// TwinCAT 3 PLC project RRP_Palletizer_Project
// ProgramVersion: 3.1.4023.0
// libraries:
//   Tc2_Standard, * (Beckhoff Automation GmbH)
//   Tc2_System, * (Beckhoff Automation GmbH)
//   Tc3_Module, * (Beckhoff Automation GmbH)
// project tree:
//   DUTs/ stMachineState.TcDUT, stMotor.TcDUT, stPneumatic1.TcDUT, stPneumatic2.TcDUT
//   GVLs/ Data_GVL.TcGVL, HMI_GVL.TcGVL, InputOutput_GVL.TcGVL
//   / BoxTask.TcTTO
//   POUs/S01_Box/ EM01_BoxShorting.TcPOU, UN01_StateMachineBox.TcPOU
//   POUs/S02_Pallet/ EM01_Dispenser.TcPOU, EM02_Shuttle.TcPOU, EM03_PalletOutfeed.TcPOU, UN01_StateMachinePallet.TcPOU
//   POUs/S03_Robot_1/ EM03_PlacingArea_2.TcPOU, EM04_PlacingArea_3.TcPOU, EM05_PlacingArea_4.TcPOU, EM01_BoxInfeed.TcPOU, EM02_PlacingArea_1.TcPOU, EM06_Robot.TcPOU, UN01_StateMachineRobot_1.TcPOU
//   POUs/Functions Blocks/ BLINK.TcPOU, FB_StateManager.TcPOU, MotorManagement.TcPOU, Pneumatic_1Coil_Management.TcPOU, Pneumatic_2Coil_Management.TcPOU
// real-time tasks:
//   TASK PlcTask: cycle T#10ms, priority 20, ADS port 350
//   TASK Box: cycle T#10ms, priority 21, ADS port 351

CONFIGURATION RRP_Palletizer_Project
    RESOURCE PLC ON TwinCAT3
        TASK BoxTask(INTERVAL := T#10ms, PRIORITY := 21);
        PROGRAM UN01_StateMachineBox WITH BoxTask : UN01_StateMachineBox;
        PROGRAM EM01_BoxShorting WITH BoxTask : EM01_BoxShorting;
    END_RESOURCE
END_CONFIGURATION

// ---- DUTs/stMachineState.TcDUT
TYPE stMachineState :
STRUCT
	Error 		: BOOL;
	CheckSafety	: BOOL;
	Aborted		: BOOL;
	Initialize	: BOOL;
	CheckToRun	: BOOL;
	Ready		: BOOL;
	Running		: BOOL;
	Stopped		: BOOL;
	ManualMode	: BOOL;
END_STRUCT
END_TYPE

// ---- DUTs/stMotor.TcDUT
TYPE stMotor :	
STRUCT
	Name				: STRING;
	TestModeActive		: BOOL;
	UseReverse			: BOOL;
	iTestForward		: BOOL;
	iTestReverse		: BOOL;
	oMoveForward		: BOOL;
	oMoveReverse		: BOOL;
	oResetError			: BOOL;
	Status_MotorRunning	: BOOL;
	Status_Error		: BOOL;
	ErrorID				: UINT;
END_STRUCT
END_TYPE

// ---- DUTs/stPneumatic1.TcDUT
TYPE stPneumatic1 : //v1.0
// UDT untuk merepresentasikan faceplate pneumatic valve 1 coil
//	Changelog:
	(* 
	v1.0 [27.12.2021] Start development UDT - Fabrilian Asali	*)	


STRUCT
	Name: STRING;
	
	TestModeActive: BOOL;
	iTest: BOOL;
	
	iSensorRetract: BOOL;
	iSensorAdvanced: BOOL;
	
	oPneumatic: BOOL;
	
	Trigger_Retract: BOOL;
	Trigger_Advanced: BOOL;
	FB_DoneRetract: BOOL;
	FB_DoneAdvanced: BOOL;
	
	Error_Retract: BOOL;
	Error_Advanced: BOOL;
END_STRUCT
END_TYPE

// ---- DUTs/stPneumatic2.TcDUT
TYPE stPneumatic2 :	//v1.0
// UDT untuk merepresentasikan faceplate pneumatic valve 1 coil
//	Changelog:
	(* 
	v1.0 [27.12.2021] Start development UDT - Fabrilian Asali	*)	

STRUCT
	Name: STRING;
	
	TestModeActive: BOOL;
	iTestRetract: BOOL;
	iTestAdvanced: BOOL;
	
	iSensorRetract: BOOL;
	iSensorAdvanced: BOOL;
	
	oPneumaticRetract: BOOL;
	oPneumaticAdvanced: BOOL;
	
	Trigger_Retract: BOOL;
	Trigger_Advanced: BOOL;
	FB_DoneRetract: BOOL;
	FB_DoneAdvanced: BOOL;
	
	Error_Retract: BOOL;
	Error_Advanced: BOOL;
END_STRUCT
END_TYPE

// ---- GVLs/Data_GVL.TcGVL
{attribute 'qualified_only'}
VAR_GLOBAL
	
//-----Box----	
	//Shorting
	StateMachineShorting			: stMachineState;
	StateMachineShorting_Error		: BOOL;
	StateMachineShorting_ErrorMsg	: STRING;
	StateMachineShorting_stsMachine	: STRING;
	bFL_StartShorting				: BOOL;
	bFL_StopShorting				: BOOL;
	bFL_ResetShorting				: BOOL;
	bFL_AckShorting					: BOOL;
	bFL_MachineErrorShorting		: BOOL;
	bFL_AutoManuaModeShorting		: BOOL;
	
//-----Pallet----		
	//Dispenser
	StateMachineDispenser			: stMachineState;
	StateMachineDispenser_Error		: BOOL;
	StateMachineDispenser_ErrorMsg	: STRING;
	StateMachineDispenser_stsMachine: STRING;
	bFL_StartDispenser				: BOOL;
	bFL_StopDispenser				: BOOL;
	bFL_ResetDispenser				: BOOL;
	bFL_AckDispenser				: BOOL;
	bFL_MachineErrorDispenser		: BOOL;
	bFL_AutoManuaModeDispenser		: BOOL;
	//Shuttle
	StateMachineShuttle				: stMachineState;
	StateMachineShuttle_Error		: BOOL;
	StateMachineShuttle_ErrorMsg	: STRING;
	StateMachineShuttle_stsMachine	: STRING;
	bFL_StartShuttle				: BOOL;
	bFL_StopShuttle					: BOOL;
	bFL_ResetShuttle				: BOOL;
	bFL_AckShuttle					: BOOL;
	bFL_MachineErrorShuttle			: BOOL;
	bFL_AutoManuaModeShuttle		: BOOL;
	//Outfeed
	StateMachineOutfeed				: stMachineState;
	StateMachineOutfeed_Error		: BOOL;
	StateMachineOutfeed_ErrorMsg	: STRING;
	StateMachineOutfeed_stsMachine	: STRING;
	bFL_StartOutfeed				: BOOL;
	bFL_StopOutfeed					: BOOL;
	bFL_ResetOutfeed				: BOOL;
	bFL_AckOutfeed					: BOOL;
	bFL_MachineErrorOutfeed			: BOOL;
	bFL_AutoManuaModeOutfeed		: BOOL;
	
//-----Robot----		
	//Infeed
	StateMachineInfeed				: stMachineState;
	StateMachineInfeed_Error		: BOOL;
	StateMachineInfeed_ErrorMsg		: STRING;
	StateMachineInfeed_stsMachine	: STRING;
	bFL_StartInfeed					: BOOL;
	bFL_StopInfeed					: BOOL;
	bFL_ResetInfeed					: BOOL;
	bFL_AckInfeed					: BOOL;
	bFL_MachineErrorInfeed			: BOOL;
	bFL_AutoManuaModeInfeed			: BOOL;	
	//Placing_1
	StateMachinePlacing_1			: stMachineState;
	StateMachinePlacing_1_Error		: BOOL;
	StateMachinePlacing_1_ErrorMsg	: STRING;
	StateMachinePlacing_1_stsMachine: STRING;
	bFL_StartPlacing_1				: BOOL;
	bFL_StopPlacing_1				: BOOL;
	bFL_ResetPlacing_1				: BOOL;
	bFL_AckPlacing_1				: BOOL;
	bFL_MachineErrorPlacing_1		: BOOL;
	bFL_AutoManuaModePlacing_1		: BOOL;
	//Placing_2
	StateMachinePlacing_2			: stMachineState;
	StateMachinePlacing_2_Error		: BOOL;
	StateMachinePlacing_2_ErrorMsg	: STRING;
	StateMachinePlacing_2_stsMachine: STRING;
	bFL_StartPlacing_2				: BOOL;
	bFL_StopPlacing_2				: BOOL;
	bFL_ResetPlacing_2				: BOOL;
	bFL_AckPlacing_2				: BOOL;
	bFL_MachineErrorPlacing_2		: BOOL;
	bFL_AutoManuaModePlacing_2		: BOOL;
	//Placing_3
	StateMachinePlacing_3			: stMachineState;
	StateMachinePlacing_3_Error		: BOOL;
	StateMachinePlacing_3_ErrorMsg	: STRING;
	StateMachinePlacing_3_stsMachine: STRING;
	bFL_StartPlacing_3				: BOOL;
	bFL_StopPlacing_3				: BOOL;
	bFL_ResetPlacing_3				: BOOL;
	bFL_AckPlacing_3				: BOOL;
	bFL_MachineErrorPlacing_3		: BOOL;
	bFL_AutoManuaModePlacing_3		: BOOL;
	//Placing_4
	StateMachinePlacing_4			: stMachineState;
	StateMachinePlacing_4_Error		: BOOL;
	StateMachinePlacing_4_ErrorMsg	: STRING;
	StateMachinePlacing_4_stsMachine: STRING;
	bFL_StartPlacing_4				: BOOL;
	bFL_StopPlacing_4				: BOOL;
	bFL_ResetPlacing_4				: BOOL;
	bFL_AckPlacing_4				: BOOL;
	bFL_MachineErrorPlacing_4		: BOOL;
	bFL_AutoManuaModePlacing_4		: BOOL;
	//Robot
	StateMachineRobot				: stMachineState;
	StateMachineRobot_Error			: BOOL;
	StateMachineRobot_ErrorMsg		: STRING;
	StateMachineRobot_stsMachine	: STRING;
	bFL_StartRobot		 			: BOOL;
	bFL_StopRobot					: BOOL;
	bFL_ResetRobot					: BOOL;
	bFL_AckRobot					: BOOL;
	bFL_MachineErrorRobot			: BOOL;
	bFL_AutoManuaModeRobot			: BOOL;
	
	bStartButton 					: BOOL;
	bStopButton 					: BOOL;
	bResetButton 					: BOOL;
	bAckButton 						: BOOL;
	bEmergencyStop 					: BOOL;
END_VAR

// ---- GVLs/HMI_GVL.TcGVL
{attribute 'qualified_only'}
VAR_GLOBAL
//-----Box----
	//Shorting
	bTestModeEnableShorting	: BOOL;
	bStartButtonShorting	: BOOL;
	bStopButtonShorting		: BOOL;
	bResetButtonShorting	: BOOL;

//-----Pallet----
	//Dispenser
	bTestModeEnableDispenser: BOOL;
	bStartButtonDispenser	: BOOL;
	bStopButtonDispenser	: BOOL;
	bResetButtonDispenser	: BOOL;
	//Outfeed
	bTestModeEnableOutfeed	: BOOL;
	bStartButtonOutfeed		: BOOL;
	bStopButtonOutfeed		: BOOL;
	bResetButtonOutfeed		: BOOL;
	//Shuttle
	bTestModeEnableShuttle	: BOOL;
	bStartButtonShuttle		: BOOL;
	bStopButtonShuttle		: BOOL;
	bResetButtonShuttle		: BOOL;

//-----Robot----
	//Infeed
	bTestModeEnableInfeed	: BOOL;
	bStartButtonInfeed		: BOOL;
	bStopButtonInfeed		: BOOL;
	bResetButtonInfeed		: BOOL;
	//Placing_1
	bTestModeEnablePlacing_1: BOOL;
	bStartButtonPlacing_1	: BOOL;
	bStopButtonPlacing_1	: BOOL;
	bResetButtonPlacing_1	: BOOL;
	//Placing_2
	bTestModeEnablePlacing_2: BOOL;
	bStartButtonPlacing_2	: BOOL;
	bStopButtonPlacing_2	: BOOL;
	bResetButtonPlacing_2	: BOOL;
	//Placing_3
	bTestModeEnablePlacing_3: BOOL;
	bStartButtonPlacing_3	: BOOL;
	bStopButtonPlacing_3	: BOOL;
	bResetButtonPlacing_3	: BOOL;
	//Placing_4
	bTestModeEnablePlacing_4: BOOL;
	bStartButtonPlacing_4	: BOOL;
	bStopButtonPlacing_4	: BOOL;
	bResetButtonPlacing_4	: BOOL;
	//Robot
	bTestModeEnableRobot	: BOOL;
	bStartButtonRobot		: BOOL;
	bStopButtonRobot		: BOOL;
	bResetButtonRobot		: BOOL;
END_VAR

// ---- GVLs/InputOutput_GVL.TcGVL
{attribute 'qualified_only'}
VAR_GLOBAL
	//Panel 1
	//Digital Input 16 Point EL1809
	xIn1000				AT 		%I*			: BOOL;		// Push Button Run at Main Panel
	xIn1001				AT 		%I*			: BOOL;		// Push Button Stop at Main Panel
	xIn1002				AT 		%I*			: BOOL;		// Push Button Alarm Reset at Main Panel
	xIn1003				AT 		%I*			: BOOL;		// Push Button Acknowledge at Main Panel
	xIn1004				AT 		%I*			: BOOL;		// Auto/Manual Mode at Main Panel
	xIn1005				AT 		%I*			: BOOL;		// Emergency Stop at Main Panel
	xIn1006				AT 		%I*			: BOOL;		//	
	xIn1007				AT 		%I*			: BOOL;		//
	xIn1008				AT 		%I*			: BOOL;		//
	xIn1009				AT 		%I*			: BOOL;		//
	xIn1010				AT 		%I*			: BOOL;		//
	xIn1011				AT 		%I*			: BOOL;		//
	xIn1012				AT 		%I*			: BOOL;		//
	xIn1013				AT 		%I*			: BOOL;		//
	xIn1014				AT 		%I*			: BOOL;		//
	xIn1015				AT 		%I*			: BOOL;		// Pressure Switch
	//Digital Input 16 Point EL1809
	xIn1100				AT 		%I*			: BOOL;		// Feedback Barcoder Reading Conveyor is Running
	xIn1101				AT 		%I*			: BOOL;		// Feedback Box Infeed Roller Conveyor 1 is Running
	xIn1102				AT 		%I*			: BOOL;		// Feedback Box Infeed Roller Conveyor 2 is Running 
	xIn1103				AT 		%I*			: BOOL;		// Feedback Box Infeed Roller Conveyor 3 is Running
	xIn1104				AT 		%I*			: BOOL;		// Feedback Box Buffer Roller Conveyor 1 is Running
	xIn1105				AT 		%I*			: BOOL;		// Feedback Box Buffer Roller Conveyor 2 is Running
	xIn1106				AT 		%I*			: BOOL;		// Feedback Box Stop & Go Belt Conveyor is Running
	xIn1107				AT 		%I*			: BOOL;		// Feedback Box Picking Roller Conveyor is Running
	xIn1108				AT 		%I*			: BOOL;		//
	xIn1109				AT 		%I*			: BOOL;		//
	xIn1110				AT 		%I*			: BOOL;		//
	xIn1111				AT 		%I*			: BOOL;		//
	xIn1112				AT 		%I*			: BOOL;		//
	xIn1113				AT 		%I*			: BOOL;		//
	xIn1114				AT 		%I*			: BOOL;		//
	xIn1115				AT 		%I*			: BOOL;		// 
	//Digital Input 16 Point EL1809
	xIn1200				AT 		%I*			: BOOL;		// RSW to Check Pneu Box Pusher for Reject Barcode when Rtc
	xIn1201				AT 		%I*			: BOOL;		// RSW to Check Pneu Box Pusher for Reject Barcode when Adv
	xIn1202				AT 		%I*			: BOOL;		// RSW to Check Pneu Box Pusher for Reject Weight when Rtc
	xIn1203				AT 		%I*			: BOOL;		// RSW to Check Pneu Box Pusher for Reject Weight when Adv
	xIn1204				AT 		%I*			: BOOL;		// RSW to Check Pneu Box Pusher when Rtc
	xIn1205				AT 		%I*			: BOOL;		// RSW to Check Pneu Box Pusher when Adv
	xIn1206				AT 		%I*			: BOOL;		//	
	xIn1207				AT 		%I*			: BOOL;		//
	xIn1208				AT 		%I*			: BOOL;		//
	xIn1209				AT 		%I*			: BOOL;		//
	xIn1210				AT 		%I*			: BOOL;		//
	xIn1211				AT 		%I*			: BOOL;		//
	xIn1212				AT 		%I*			: BOOL;		//
	xIn1213				AT 		%I*			: BOOL;		//
	xIn1214				AT 		%I*			: BOOL;		//
	xIn1215				AT 		%I*			: BOOL;		// 
	//Digital Input 16 Point EL1809
	xIn1300				AT 		%I*			: BOOL;		// PSR Back to Detect Box at Barcoder Reading Conv
	xIn1301				AT 		%I*			: BOOL;		// PSR Middle to Detect Box at Barcoder Reading Conv
	xIn1302				AT 		%I*			: BOOL;		// PSR Front to Detect Box at Barcoder Reading Conv
	xIn1303				AT 		%I*			: BOOL;		// PSR to Detect Box at Outfeed Check Weigher
	xIn1304				AT 		%I*			: BOOL;		// PSR to Detect Box at Reject Barcode
	xIn1305				AT 		%I*			: BOOL;		// PSR to Detect Box at Reject Weight
	xIn1306				AT 		%I*			: BOOL;		// PSR to Detect Box for Buffer at Infeed Roller Conv
	xIn1307				AT 		%I*			: BOOL;		// PSR to Detect Box for Pusher at Infeed Roller Conv
	xIn1308				AT 		%I*			: BOOL;		// PSR to Detect Box at Buffer Roller Conv 1
	xIn1309				AT 		%I*			: BOOL;		// PSR to Detect Box at Buffer Roller Conv 2
	xIn1310				AT 		%I*			: BOOL;		// PSR to Detect Box at Stop & Go Belt Conv
	xIn1311				AT 		%I*			: BOOL;		// PSR to Detect Box at Picking Conv
	xIn1312				AT 		%I*			: BOOL;		// PSR to Detect Box at Gravity Roller Conv
	xIn1313				AT 		%I*			: BOOL;		// PSR to Detect Box at Gravity Roller Conv
	xIn1314				AT 		%I*			: BOOL;		// PSR to Detect Box at Gravity Roller Conv Reject
	xIn1315				AT 		%I*			: BOOL;		// PSR to Detect Box at Gravity Roller Conv Reject
	//Safety Input SI 4 Point EL1904
	xsIn1400			AT 		%I*			: BOOL;		// Emergency Stop Channel 1 at Main Panel
	xsIn1402			AT 		%I*			: BOOL;		// Emergency Stop Channel 2 at Main Panel
	xsIn1404			AT 		%I*			: BOOL;		// Auto Machine at Main Panel
	xsIn1406			AT 		%I*			: BOOL;		// Manual Machine at Main Panel
	//Panel 2
	//Digital Input 16 Point EL1809
	xIn3000				AT 		%I*			: BOOL;		//Push Button Run at P2
	xIn3001				AT 		%I*			: BOOL;		// Push Button Stop at P2
	xIn3002				AT 		%I*			: BOOL;		// Push Button Alarm Reset at P2
	xIn3003				AT 		%I*			: BOOL;		// Emergency Stop at P2
	xIn3004				AT 		%I*			: BOOL;		// Push Button Run at Dispenser
	xIn3005				AT 		%I*			: BOOL;		// Push Button Stop at Dispenser
	xIn3006				AT 		%I*			: BOOL;		// Push Button Alarm Reset at Dispenser
	xIn3007				AT 		%I*			: BOOL;		// Push Button Acknowledge at Dispenser
	xIn3008				AT 		%I*			: BOOL;		// Auto/Manual Switch at Dispenser
	xIn3009				AT 		%I*			: BOOL;		// Emergency Stop at Dispenser
	xIn3010				AT 		%I*			: BOOL;		// Manual Switch For Test Pneumatic Vertical UP
	xIn3011				AT 		%I*			: BOOL;		// Manual Switch For Test Pneumatic Vertical DOWN
	xIn3012				AT 		%I*			: BOOL;		// Manual Switch for Test Pneumatic Horizontal
	xIn3013				AT 		%I*			: BOOL;		// Manual Switch for Test Motor Empty Stacks Pallet Infeed Roller Conv
	xIn3014				AT 		%I*			: BOOL;		// Manual Switch for Test Motor Automatic Pallet Roller Conv
	xIn3015				AT 		%I*			: BOOL;		// Pressure Switch for Pallet Dispenser
	//Digital Input 16 Point EL1809
	xIn3100				AT 		%I*			: BOOL;		// Feedback Empty stacks pallet infeed roller conv is Running
	xIn3101				AT 		%I*			: BOOL;		// Feedback Automatic pallet roller conv is Running
	xIn3102				AT 		%I*			: BOOL;		// Feedback Box placing at pallet roller conv L1 is Running
	xIn3103				AT 		%I*			: BOOL;		// Feedback Box placing at pallet roller conv L2 is Running
	xIn3104				AT 		%I*			: BOOL;		// Feedback Box placing at pallet roller conv L3 is Running
	xIn3105				AT 		%I*			: BOOL;		// Feedback Box placing at pallet roller conv L4 is Running
	xIn3106				AT 		%I*			: BOOL;		// Feedback  Empty & Load pallet transfer roller conv is Running
	xIn3107				AT 		%I*			: BOOL;		// Feedback Empty & Loaded pallet turning conv 1 is Running
	xIn3108				AT 		%I*			: BOOL;		// Feedback Empty & Loaded pallet turning conv 2 is Running
	xIn3109				AT 		%I*			: BOOL;		// Feedback Loaded Pallet buffer roller conv before Wrapping is Running
	xIn3110				AT 		%I*			: BOOL;		// Feedback Loaded Pallet buffer roller conv after Wrapping is Running
	xIn3111				AT 		%I*			: BOOL;		// Feedback Loaded pallet outfeed roller conv is Running
	xIn3112				AT 		%I*			: BOOL;		// 
	xIn3113				AT 		%I*			: BOOL;		// 
	xIn3114				AT 		%I*			: BOOL;		// 
	xIn3115				AT 		%I*			: BOOL;		// 
	//Digital Input 16 Point EL1809
	xIn3200				AT 		%I*			: BOOL;		// PSR Back at Placing Conv L1
	xIn3201				AT 		%I*			: BOOL;		// PSR Front at Placing Conv L1
	xIn3202				AT 		%I*			: BOOL;		// PSR Back at Placing Conv L2
	xIn3203				AT 		%I*			: BOOL;		// PSR Front at Placing Conv L2
	xIn3204				AT 		%I*			: BOOL;		// PSR Back at Placing Conv L3
	xIn3205				AT 		%I*			: BOOL;		// PSR Front at Placing Conv L3
	xIn3206				AT 		%I*			: BOOL;		// PSR Back at Placing Conv L4
	xIn3207				AT 		%I*			: BOOL;		// PSR Front at Placing Conv L4
	xIn3208				AT 		%I*			: BOOL;		// PSR Back at Empty & Load pallet transfer roller conv L4
	xIn3209				AT 		%I*			: BOOL;		// PSR Front at Empty & Load pallet transfer roller conv L4
	xIn3210				AT 		%I*			: BOOL;		// PSR Back at Empty & Loaded pallet turning conv
	xIn3211				AT 		%I*			: BOOL;		// PSR Front at Empty & Loaded pallet turning conv
	xIn3212				AT 		%I*			: BOOL;		// PSR Back at Loaded Pallet buffer roller conv before Wrapping
	xIn3213				AT 		%I*			: BOOL;		// PSR Front at Loaded Pallet buffer roller conv before Wrapping
	xIn3214				AT 		%I*			: BOOL;		// PSR Back at Loaded Pallet buffer roller conv after Wrapping
	xIn3215				AT 		%I*			: BOOL;		// PSR Front at Loaded Pallet buffer roller conv after Wrapping
	//Digital Input 16 Point EL1809
	xIn3300				AT 		%I*			: BOOL;		// PSR Back at Loaded pallet outfeed roller conv
	xIn3301				AT 		%I*			: BOOL;		// PSR Front at Loaded pallet outfeed roller conv
	xIn3302				AT 		%I*			: BOOL;		// 
	xIn3303				AT 		%I*			: BOOL;		// 
	xIn3304				AT 		%I*			: BOOL;		// 
	xIn3305				AT 		%I*			: BOOL;		// 
	xIn3306				AT 		%I*			: BOOL;		// 
	xIn3307				AT 		%I*			: BOOL;		// 
	xIn3308				AT 		%I*			: BOOL;		// PRX 1 at Empty & Loaded pallet turning conv
	xIn3309				AT 		%I*			: BOOL;		// PRX 2 at Empty & Loaded pallet turning conv
	xIn3310				AT 		%I*			: BOOL;		// PRX 3 at Empty & Loaded pallet turning conv
	xIn3311				AT 		%I*			: BOOL;		// 
	xIn3312				AT 		%I*			: BOOL;		// 
	xIn3313				AT 		%I*			: BOOL;		// 
	xIn3314				AT 		%I*			: BOOL;		// 
	xIn3315				AT 		%I*			: BOOL;		// 
	//Digital Input 16 Point EL1809
	xIn3400				AT 		%I*			: BOOL;		// PSR to Check Back Pallet at Empty stacks pallet infeed roller conv
	xIn3401				AT 		%I*			: BOOL;		// PSR to Check Front Pallet at Empty stacks pallet infeed roller conv
	xIn3402				AT 		%I*			: BOOL;		// PSR to Check Back Pallet at Automatic pallet roller conv
	xIn3403				AT 		%I*			: BOOL;		// PSR to Check Front Pallet at Automatic pallet roller conv
	xIn3404				AT 		%I*			: BOOL;		// PSR to Check Stack Pallet at Automatic pallet roller conv
	xIn3405				AT 		%I*			: BOOL;		// RSW to Check Right Pneumatic Horizontal When Retract
	xIn3406				AT 		%I*			: BOOL;		// RSW to Check Right Pneumatic Horizontal When Advanced
	xIn3407				AT 		%I*			: BOOL;		// RSW to Check Left Pneumatic Horizontal When Retract
	xIn3408				AT 		%I*			: BOOL;		// RSW to Check Left Pneumatic Horizontal When Advanced
	xIn3409				AT 		%I*			: BOOL;		// Proximity Sensor at Retract Position Left Pneumatic Vertical
	xIn3410				AT 		%I*			: BOOL;		// PRX at Middle Position Left Pneumatic Vertical
	xIn3411				AT 		%I*			: BOOL;		// PRX at Advanced Position Left Pneumatic Vertical
	xIn3412				AT 		%I*			: BOOL;		// PRX at Retract Position Right Pneumatic Vertical
	xIn3413				AT 		%I*			: BOOL;		// PRX at Middle Position Right Pneumatic Vertical
	xIn3414				AT 		%I*			: BOOL;		// PRX at Advanced Position Right Pneumatic Vertical
	xIn3415				AT 		%I*			: BOOL;		// 
	//Digital Input 16 Point EL1809
	xIn3500				AT 		%I*			: BOOL;		// 
	xIn3501				AT 		%I*			: BOOL;		// 
	xIn3502				AT 		%I*			: BOOL;		// 
	xIn3503				AT 		%I*			: BOOL;		// 
	xIn3504				AT 		%I*			: BOOL;		// 
	xIn3505				AT 		%I*			: BOOL;		// 
	xIn3506				AT 		%I*			: BOOL;		// 
	xIn3507				AT 		%I*			: BOOL;		// 
	xIn3508				AT 		%I*			: BOOL;		// 
	xIn3509				AT 		%I*			: BOOL;		// 
	xIn3510				AT 		%I*			: BOOL;		// 
	xIn3511				AT 		%I*			: BOOL;		// 
	xIn3512				AT 		%I*			: BOOL;		// 
	xIn3513				AT 		%I*			: BOOL;		// 
	xIn3514				AT 		%I*			: BOOL;		// 
	xIn3515				AT 		%I*			: BOOL;		// 
	//Safety Input SI 4 Point EL1904
	xsIn3600			AT 		%I*			: BOOL;		// Emergency Stop at Channel 1
	xsIn3602			AT 		%I*			: BOOL;		// Emergency Stop at Channel 2
	xsIn3604			AT 		%I*			: BOOL;		// Safety Door Solenoid Channel 1
	xsIn3606			AT 		%I*			: BOOL;		// Safety Door Solenoid Channel 2
	//Safety Input SI 4 Point EL1904
	xsIn3700			AT 		%I*			: BOOL;		// Light Curtain Channel 1 at Dispenser
	xsIn3702			AT 		%I*			: BOOL;		// Light Curtain Channel 2 at Dispenser
	xsIn3704			AT 		%I*			: BOOL;		// Light Curtain Channel 1 at Loaded Outfeed
	xsIn3706			AT 		%I*			: BOOL;		// Light Curtain Channel 2 at Loaded Outfeed
	//Panel 3
	//Digital Input 16 Point EL1809
	xIn5000				AT 		%I*			: BOOL;		// Feedback Empty pallet shuttle is Running
	xIn5001				AT 		%I*			: BOOL;		// Feedback Load pallet shuttle is Running
	xIn5002				AT 		%I*			: BOOL;		// Feedback Drive Shuttle is Running
	xIn5003				AT 		%I*			: BOOL;		// 
	xIn5004				AT 		%I*			: BOOL;		// PSR To Detect Front Pallet at Empty Pallet Shuttle
	xIn5005				AT 		%I*			: BOOL;		// PSR To Detect Back Pallet at Empty Pallet Shuttle
	xIn5006				AT 		%I*			: BOOL;		// PSR To Detect End Of Front Pallet at Empty Pallet Shuttle
	xIn5007				AT 		%I*			: BOOL;		// PSR To Detect End Of Back Pallet at Empty Pallet Shuttle
	xIn5008				AT 		%I*			: BOOL;		// PSR To Detect Front Pallet at Load Pallet Shuttle
	xIn5009				AT 		%I*			: BOOL;		// PSR To Detect Back Pallet at Load Pallet Shuttle
	xIn5010				AT 		%I*			: BOOL;		// PSR To Detect End Of Front Pallet at Load Pallet Shuttle
	xIn5011				AT 		%I*			: BOOL;		// PSR To Detect End Of Back Pallet at Load Pallet Shuttle
	xIn5012				AT 		%I*			: BOOL;		// Limit Switch To Detect Left Limit Area
	xIn5013				AT 		%I*			: BOOL;		// Limit Switch To Detect Right Limit Area
	xIn5014				AT 		%I*			: BOOL;		// PRX to Detect Left Limit Area
	xIn5015				AT 		%I*			: BOOL;		// PRX to Detect Right Limit Area
	//Gripper Robot
	//Digital Input 16 Point
	xIn_0				AT 		%I*			: BOOL;		// RSW to Check Open Claw Box
	xIn_1				AT 		%I*			: BOOL;		// RSW to Check Close Claw Box
	xIn_2				AT 		%I*			: BOOL;		// RSW to Check Open Clamping Box
	xIn_3				AT 		%I*			: BOOL;		// RSW to Check Close Clamping Box
	xIn_4				AT 		%I*			: BOOL;		// PSR to Check Box at Gripper
	xIn_5				AT 		%I*			: BOOL;		// 
	xIn_6				AT 		%I*			: BOOL;		// 
	xIn_7				AT 		%I*			: BOOL;		// 
	xIn_8				AT 		%I*			: BOOL;		// 
	xIn_9				AT 		%I*			: BOOL;		// 
	xIn_10				AT 		%I*			: BOOL;		// 
	xIn_11				AT 		%I*			: BOOL;		// 
	xIn_12				AT 		%I*			: BOOL;		// 
	xIn_13				AT 		%I*			: BOOL;		// 
	xIn_14				AT 		%I*			: BOOL;		// 
	xIn_15				AT 		%I*			: BOOL;		// 
	//Panel 1
	//Digital Output 16 Point EL2809
	xOut2000			AT 		%Q*			: BOOL;		// Indicator Machine Running at Main Panel
	xOut2001			AT 		%Q*			: BOOL;		// Indicator Machine Error at Main Panel
	xOut2002			AT 		%Q*			: BOOL;		// Indicator Acknowledge at Main Panel
	xOut2003			AT 		%Q*			: BOOL;		// Indicator Auto Mode
	xOut2004			AT 		%Q*			: BOOL;		// Indicator Manual Mode
	xOut2005			AT 		%Q*			: BOOL;		// Indicator Tower Lamp Red
	xOut2006			AT 		%Q*			: BOOL;		// Indicator Tower Lamp Yellow
	xOut2007			AT 		%Q*			: BOOL;		// Indicator Tower Lamp Green
	xOut2008			AT 		%Q*			: BOOL;		// Indicator Tower Lamp Blue
	xOut2009			AT 		%Q*			: BOOL;		// Indicator Buzzer
	xOut2010			AT 		%Q*			: BOOL;		//
	xOut2011			AT 		%Q*			: BOOL;		//
	xOut2012			AT 		%Q*			: BOOL;		//
	xOut2013			AT 		%Q*			: BOOL;		//
	xOut2014			AT 		%Q*			: BOOL;		//
	xOut2015			AT 		%Q*			: BOOL;		// 
	//Digital Output 16 Point EL2809
	xOut2100			AT 		%Q*			: BOOL;		// Move Forward for Barcoder Reading Conveyor
	xOut2101			AT 		%Q*			: BOOL;		// Move Forward for Box Infeed Roller Conveyor 1
	xOut2102			AT 		%Q*			: BOOL;		// Move Forward for Box Infeed Roller Conveyor 2
	xOut2103			AT 		%Q*			: BOOL;		// Move Forward for Box Infeed Roller Conveyor 3
	xOut2104			AT 		%Q*			: BOOL;		// Move Forward for Box Buffer Roller Conveyor 1
	xOut2105			AT 		%Q*			: BOOL;		// Move Forward for Box Buffer Roller Conveyor 2
	xOut2106			AT 		%Q*			: BOOL;		// Move Forward for Box Stop & Go Belt Conveyor
	xOut2107			AT 		%Q*			: BOOL;		// Move Forward for Box Picking Roller Conveyor
	xOut2108			AT 		%Q*			: BOOL;		//
	xOut2109			AT 		%Q*			: BOOL;		//
	xOut2110			AT 		%Q*			: BOOL;		//
	xOut2111			AT 		%Q*			: BOOL;		//
	xOut2112			AT 		%Q*			: BOOL;		//
	xOut2113			AT 		%Q*			: BOOL;		//
	xOut2114			AT 		%Q*			: BOOL;		//
	xOut2115			AT 		%Q*			: BOOL;		// Reset Error for All Inverter at Main Panel, Relay
	//Digital Output 16 Point EL2809
	xOut2200			AT 		%Q*			: BOOL;		// Pneumatic Box Pusher for Reject Barcode
	xOut2201			AT 		%Q*			: BOOL;		// Pneumatic Box Pusher for Reject Weight
	xOut2202			AT 		%Q*			: BOOL;		// Pneumatic Box Pusher
	xOut2203			AT 		%Q*			: BOOL;		// 
	xOut2204			AT 		%Q*			: BOOL;		// 
	xOut2205			AT 		%Q*			: BOOL;		// 
	xOut2206			AT 		%Q*			: BOOL;		//	
	xOut2207			AT 		%Q*			: BOOL;		//
	xOut2208			AT 		%Q*			: BOOL;		//
	xOut2209			AT 		%Q*			: BOOL;		//
	xOut2210			AT 		%Q*			: BOOL;		//
	xOut2211			AT 		%Q*			: BOOL;		//
	xOut2212			AT 		%Q*			: BOOL;		//
	xOut2213			AT 		%Q*			: BOOL;		//
	xOut2214			AT 		%Q*			: BOOL;		//
	xOut2215			AT 		%Q*			: BOOL;		// 
	//Safety Output SO 4 Point EL2904
	xsOut2300			AT 		%Q*			: BOOL;		// Enable STO Conveyor Channel 1
	xsOut2302			AT 		%Q*			: BOOL;		// Enable STO Conveyor Channel 2
	xsOut2304			AT 		%Q*			: BOOL;		// Enable Air Supply Channel 1
	xsOut2306			AT 		%Q*			: BOOL;		// Enable Air Supply Channel 2
	//Panel 2
	//Digital Output 16 Point EL2809
	xOut4000			AT 		%Q*			: BOOL;		// Indicator Machine Running at P2
	xOut4001			AT 		%Q*			: BOOL;		// Indicator Machine Error at P2
	xOut4002			AT 		%Q*			: BOOL;		// Indicator Tower Lamp Red at P2
	xOut4003			AT 		%Q*			: BOOL;		// Indicator Tower Lamp Yellow at P2
	xOut4004			AT 		%Q*			: BOOL;		// Indicator Tower Lamp Green at P2
	xOut4005			AT 		%Q*			: BOOL;		// Indicator Tower Lamp Blue at P2
	xOut4006			AT 		%Q*			: BOOL;		// Indicator Buzzer at P2
	xOut4007			AT 		%Q*			: BOOL;		// Indicator Machine Running at Dispenser
	xOut4008			AT 		%Q*			: BOOL;		// Indicator Machine Error at Dispenser
	xOut4009			AT 		%Q*			: BOOL;		// Indicator Acknowledge at Dispenser
	xOut4010			AT 		%Q*			: BOOL;		// Indicator Auto at Dispenser
	xOut4011			AT 		%Q*			: BOOL;		// Indicator Manual at Dispenser
	xOut4012			AT 		%Q*			: BOOL;		//
	xOut4013			AT 		%Q*			: BOOL;		//
	xOut4014			AT 		%Q*			: BOOL;		//
	xOut4015			AT 		%Q*			: BOOL;		// 
	//Digital Output 16 Point EL2809
	xOut4100			AT 		%Q*			: BOOL;		// Move Forward for Empty stacks pallet infeed roller conv
	xOut4101			AT 		%Q*			: BOOL;		// Move Forward for Automatic pallet roller conv
	xOut4102			AT 		%Q*			: BOOL;		// Move Forward for Box placing at pallet roller conv L1
	xOut4103			AT 		%Q*			: BOOL;		// Move Forward for Box placing at pallet roller conv L2
	xOut4104			AT 		%Q*			: BOOL;		// Move Forward for Box placing at pallet roller conv L3
	xOut4105			AT 		%Q*			: BOOL;		// Move Forward for Box placing at pallet roller conv L4
	xOut4106			AT 		%Q*			: BOOL;		// Move Forward for Empty & Load pallet transfer roller conv
	xOut4107			AT 		%Q*			: BOOL;		// Move Forward for Empty & Loaded pallet turning conv 1
	xOut4108			AT 		%Q*			: BOOL;		// Move Forward for Empty & Loaded pallet turning conv 2
	xOut4109			AT 		%Q*			: BOOL;		// Move Forward for Loaded Pallet buffer roller conv before wrapping
	xOut4110			AT 		%Q*			: BOOL;		// Move Forward for Loaded Pallet buffer roller conv. after wrapping
	xOut4111			AT 		%Q*			: BOOL;		// Move Forward for Loaded pallet outfeed roller conv
	xOut4112			AT 		%Q*			: BOOL;		//
	xOut4113			AT 		%Q*			: BOOL;		//
	xOut4114			AT 		%Q*			: BOOL;		// 
	xOut4115			AT 		%Q*			: BOOL;		// Reset Error for All Inverter at P2, Relay
	//Digital Output 16 Point EL2809
	xOut4200			AT 		%Q*			: BOOL;		// Pneumatic Vertical Up
	xOut4201			AT 		%Q*			: BOOL;		// Pneumatic Vertical Down
	xOut4202			AT 		%Q*			: BOOL;		// Pneumatic Horizontal Rectract
	xOut4203			AT 		%Q*			: BOOL;		// Pneumatic Horizontal Advanced
	xOut4204			AT 		%Q*			: BOOL;		// 
	xOut4205			AT 		%Q*			: BOOL;		// 
	xOut4206			AT 		%Q*			: BOOL;		//	
	xOut4207			AT 		%Q*			: BOOL;		//
	xOut4208			AT 		%Q*			: BOOL;		//
	xOut4209			AT 		%Q*			: BOOL;		//
	xOut4210			AT 		%Q*			: BOOL;		//
	xOut4211			AT 		%Q*			: BOOL;		//
	xOut4212			AT 		%Q*			: BOOL;		//
	xOut4213			AT 		%Q*			: BOOL;		//
	xOut4214			AT 		%Q*			: BOOL;		//
	xOut4215			AT 		%Q*			: BOOL;		// 
	//Safety Output SO 4 Point EL2904
	xsOut4300			AT 		%Q*			: BOOL;		// Enable STO Conveyor Channel 1
	xsOut4302			AT 		%Q*			: BOOL;		// Enable STO Conveyor Channel 2
	xsOut4304			AT 		%Q*			: BOOL;		// Enable Solenoid Door Coil Channel 1
	xsOut4306			AT 		%Q*			: BOOL;		// Enable Solenoid Door Coil Channel 2
	//Panel 3
	//Digital Output 16 Point EL2809
	xOut5000			AT 		%Q*			: BOOL;		// Move Forward for Empty pallet shuttle
	xOut5001			AT 		%Q*			: BOOL;		// Move Forward for Load pallet shuttle
	xOut5002			AT 		%Q*			: BOOL;		// Move Reverse for Load pallet shuttle
	xOut5003			AT 		%Q*			: BOOL;		// Move Forward for Drive Shuttle
	xOut5004			AT 		%Q*			: BOOL;		// Move Reverse for Drive Shuttle
	xOut5005			AT 		%Q*			: BOOL;		// 
	xOut5006			AT 		%Q*			: BOOL;		// 
	xOut5007			AT 		%Q*			: BOOL;		// 
	xOut5008			AT 		%Q*			: BOOL;		// 
	xOut5009			AT 		%Q*			: BOOL;		// 
	xOut5010			AT 		%Q*			: BOOL;		// 
	xOut5011			AT 		%Q*			: BOOL;		// 
	xOut5012			AT 		%Q*			: BOOL;		// 
	xOut5013			AT 		%Q*			: BOOL;		// 
	xOut5014			AT 		%Q*			: BOOL;		// 
	xOut5015			AT 		%Q*			: BOOL;		// 
	//Gripper Robot
	//Digital Output 16 Point
	xOut_0				AT 		%Q*			: BOOL;		// Pneumatic Gripper Claw Open Box
	xOut_1				AT 		%Q*			: BOOL;		// Pneumatic Gripper Claw Close Box
	xOut_2				AT 		%Q*			: BOOL;		// Pneumatic Gripper Clamping Open Box
	xOut_3				AT 		%Q*			: BOOL;		// Pneumatic Gripper Clamping Close Box
	xOut_4				AT 		%Q*			: BOOL;		// 
	xOut_5				AT 		%Q*			: BOOL;		// 
	xOut_6				AT 		%Q*			: BOOL;		// 
	xOut_7				AT 		%Q*			: BOOL;		// 
	xOut_8				AT 		%Q*			: BOOL;		// 
	xOut_9				AT 		%Q*			: BOOL;		// 
	xOut_10				AT 		%Q*			: BOOL;		// 
	xOut_11				AT 		%Q*			: BOOL;		// 
	xOut_12				AT 		%Q*			: BOOL;		// 
	xOut_13				AT 		%Q*			: BOOL;		// 
	xOut_14				AT 		%Q*			: BOOL;		// 
	xOut_15				AT 		%Q*			: BOOL;		// 
END_VAR

// ---- POUs/S01_Box/UN01_StateMachineBox.TcPOU
PROGRAM UN01_StateMachineBox
VAR
	FB_StateMachineShorting	: FB_StateManager;
END_VAR

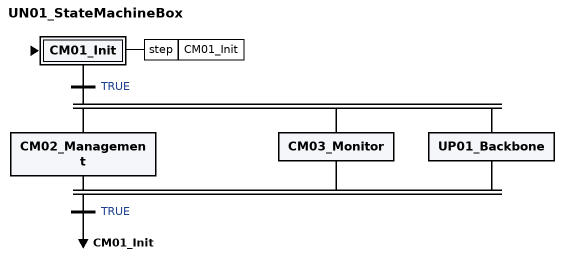
INITIAL_STEP CM01_Init:
    CM01_Init(N);  // step action
END_STEP
TRANSITION FROM CM01_Init TO (CM02_Management, CM03_Monitor, UP01_Backbone)
    := TRUE;
END_TRANSITION
STEP CM02_Management:
END_STEP
STEP CM03_Monitor:
END_STEP
STEP UP01_Backbone:
END_STEP
TRANSITION FROM (CM02_Management, CM03_Monitor, UP01_Backbone) TO CM01_Init
    := TRUE;
END_TRANSITION

ACTION CM01_Init:
//Shorting
Data_GVL.bFL_StartShorting 			:= Data_GVL.bStartButton OR HMI_GVL.bStartButtonShorting;
Data_GVL.bFL_StopShorting 			:= Data_GVL.bStopButton OR HMI_GVL.bStopButtonShorting;
Data_GVL.bFL_ResetShorting 			:= Data_GVL.bResetButton OR HMI_GVL.bResetButtonShorting;
Data_GVL.bFL_AutoManuaModeShorting 	:= NOT Data_GVL.StateMachineShorting.Running AND HMI_GVL.bTestModeEnableShorting;
END_ACTION

ACTION CM02_Management:
// NETWORK 1
END_ACTION

ACTION CM03_Monitor:
// NETWORK 1
END_ACTION

ACTION UP01_Backbone:
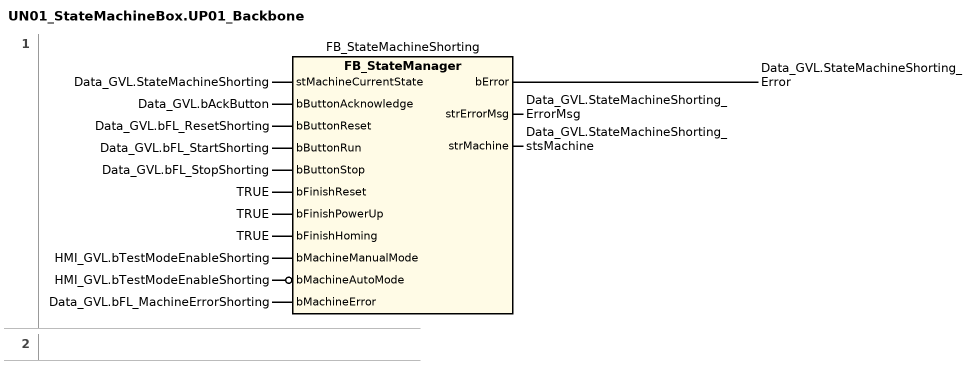
// NETWORK 1
FB_StateMachineShorting(
    stMachineCurrentState := Data_GVL.StateMachineShorting,
    bButtonAcknowledge := Data_GVL.bAckButton,
    bButtonReset := Data_GVL.bFL_ResetShorting,
    bButtonRun := Data_GVL.bFL_StartShorting,
    bButtonStop := Data_GVL.bFL_StopShorting,
    bFinishReset := TRUE,
    bFinishPowerUp := TRUE,
    bFinishHoming := TRUE,
    bMachineManualMode := HMI_GVL.bTestModeEnableShorting,
    bMachineAutoMode := NOT HMI_GVL.bTestModeEnableShorting,
    bMachineError := Data_GVL.bFL_MachineErrorShorting,
    strErrorMsg => Data_GVL.StateMachineShorting_ErrorMsg,
    strMachine => Data_GVL.StateMachineShorting_stsMachine); // FB_StateManager
Data_GVL.StateMachineShorting_Error := FB_StateMachineShorting.bError;

// NETWORK 2
END_ACTION

END_PROGRAM

// ---- POUs/Functions Blocks/FB_StateManager.TcPOU
FUNCTION_BLOCK FB_StateManager
VAR_IN_OUT
	stMachineCurrentState			: stMachineState;
END_VAR
VAR_INPUT
	bButtonAcknowledge				: BOOL;		// User Input for Error Acknowledgement
	bButtonReset					: BOOL;		// User Input for Reset 
	bButtonRun						: BOOL;		// User Input for Starting Machine Running Sequence
	bButtonStop						: BOOL;		// User Input for Stopping Machine Running Sequence
	bFinishReset					: BOOL;
	bFinishPowerUp					: BOOL;
	bFinishHoming					: BOOL;
	bMachineManualMode				: BOOL;		// Input(s) Required to Change Machine Operation Mode Into Manual Mode
	bMachineAutoMode				: BOOL;		// Input(s) Required to Change Machine Operation Mode Into Auto Mode
	bMachineError					: BOOL;		// Input(s) required to make the machine goes into error state
END_VAR
VAR_OUTPUT
	bError							: BOOL;		
	strErrorMsg						: STRING;	
	strMachine						: STRING;
END_VAR
VAR
	bFL_AutoModeActive				: BOOL;
	bFL_ManualModeActive			: BOOL;
	bInit							: BOOL;
	StateIndex						: UINT;
	bFL_Error						: BOOL;
END_VAR

//=======FB_StateManager v1.0=======
//Used UDTs: MachineState - v1.0
//
//Changelog: 
//v1.0 [15.01.2021] Start Function block development - Fabrilian Asali
//
//===================================

// FB initialization
IF NOT bInit THEN
	stMachineCurrentState.Error 		:= FALSE;
	stMachineCurrentState.CheckSafety	:= FALSE;
	stMachineCurrentState.Aborted		:= FALSE;
	stMachineCurrentState.Initialize	:= FALSE;
	stMachineCurrentState.CheckToRun	:= FALSE;
	stMachineCurrentState.Ready			:= FALSE;
	stMachineCurrentState.Running		:= FALSE;
	stMachineCurrentState.Stopped		:= FALSE;
	stMachineCurrentState.ManualMode	:= FALSE;
	bFL_Error							:= FALSE;
	StateIndex							:= 0;
	bInit								:= TRUE;
END_IF;

//Error detection logic | reset machine state to error state
IF bMachineError AND NOT bFL_Error THEN
	StateIndex 	:= 0;
	bFL_Error		:= TRUE;
END_IF;

//Special case reset trigger (direct from reset push button trigger)
IF bButtonAcknowledge THEN
	bError			:= FALSE;
	strErrorMsg	:= '';
END_IF;

//Auto Manual Mode Selection Logic
IF bMachineAutoMode AND NOT bMachineManualMode THEN
	bFL_AutoModeActive 							:= TRUE;
	bFL_ManualModeActive					 	:= FALSE;
ELSIF NOT bMachineAutoMode AND bMachineManualMode THEN
	bFL_ManualModeActive					 	:= TRUE;
	bFL_AutoModeActive 							:= FALSE;
ELSE
	bError 										:= TRUE;
	strErrorMsg 								:= 'Operation Mode Change Detected.';
	bFL_AutoModeActive 							:= FALSE;
	bFL_ManualModeActive						:= FALSE;
END_IF;

CASE StateIndex OF
	0: //Error State
		stMachineCurrentState.Error 		:= TRUE;
		stMachineCurrentState.CheckSafety	:= FALSE;
		stMachineCurrentState.Aborted		:= FALSE;
		stMachineCurrentState.Initialize	:= FALSE;
		stMachineCurrentState.CheckToRun	:= FALSE;
		stMachineCurrentState.Ready			:= FALSE;
		stMachineCurrentState.Running		:= FALSE;
		stMachineCurrentState.Stopped		:= FALSE;
		stMachineCurrentState.ManualMode	:= FALSE;
		strMachine							:= 'Error';
		IF bButtonAcknowledge THEN		
			StateIndex := 10;
		END_IF;
	
	10: //CheckSafety State
		stMachineCurrentState.Error 		:= FALSE;
		stMachineCurrentState.CheckSafety	:= TRUE;
		stMachineCurrentState.Aborted		:= FALSE;
		stMachineCurrentState.Initialize	:= FALSE;
		stMachineCurrentState.CheckToRun	:= FALSE;
		stMachineCurrentState.Ready			:= FALSE;
		stMachineCurrentState.Running		:= FALSE;
		stMachineCurrentState.Stopped		:= FALSE;
		stMachineCurrentState.ManualMode	:= FALSE;
		strMachine							:= 'Safety';
		IF NOT bMachineError THEN		
			StateIndex 	:= 20;
			bFL_Error		:= FALSE;
		ELSE
			bError 			:= TRUE;
			strErrorMsg := 'Machine Check Safety Failed';
			StateIndex	:= 0;
		END_IF;	

	20: //Aborted State | auto manual mode branching
		stMachineCurrentState.Error 		:= FALSE;
		stMachineCurrentState.CheckSafety	:= FALSE;
		stMachineCurrentState.Aborted		:= TRUE;
		stMachineCurrentState.Initialize	:= FALSE;
		stMachineCurrentState.CheckToRun	:= FALSE;
		stMachineCurrentState.Ready			:= FALSE;
		stMachineCurrentState.Running		:= FALSE;
		stMachineCurrentState.Stopped		:= FALSE;
		stMachineCurrentState.ManualMode	:= FALSE;
		strMachine							:= 'Aborted';		
		IF bFL_AutoModeActive AND bButtonReset THEN
			StateIndex := 30;
		ELSIF bFL_ManualModeActive THEN
			StateIndex := 1000;
		END_IF;

	30: //Initialize State
		stMachineCurrentState.Error 		:= FALSE;
		stMachineCurrentState.CheckSafety	:= FALSE;
		stMachineCurrentState.Aborted		:= FALSE;
		stMachineCurrentState.Initialize	:= TRUE;
		stMachineCurrentState.CheckToRun	:= FALSE;
		stMachineCurrentState.Ready			:= FALSE;
		stMachineCurrentState.Running		:= FALSE;
		stMachineCurrentState.Stopped		:= FALSE;
		stMachineCurrentState.ManualMode	:= FALSE;
		strMachine							:= 'Initialize';				
		IF bFinishReset AND bFinishPowerUp THEN
			StateIndex := 40;
		END_IF;
		
	40: //CheckToRun State
		stMachineCurrentState.Error 		:= FALSE;
		stMachineCurrentState.CheckSafety	:= FALSE;
		stMachineCurrentState.Aborted		:= FALSE;
		stMachineCurrentState.Initialize	:= FALSE;
		stMachineCurrentState.CheckToRun	:= TRUE;
		stMachineCurrentState.Ready			:= FALSE;
		stMachineCurrentState.Running		:= FALSE;
		stMachineCurrentState.Stopped		:= FALSE;
		stMachineCurrentState.ManualMode	:= FALSE;
		strMachine							:= 'Check Run';		
		IF bFinishHoming THEN
			StateIndex := 50;
		END_IF;
		
	50: //Ready State
		stMachineCurrentState.Error 		:= FALSE;
		stMachineCurrentState.CheckSafety	:= FALSE;
		stMachineCurrentState.Aborted		:= FALSE;
		stMachineCurrentState.Initialize	:= FALSE;
		stMachineCurrentState.CheckToRun	:= FALSE;
		stMachineCurrentState.Ready			:= TRUE;
		stMachineCurrentState.Running		:= FALSE;
		stMachineCurrentState.Stopped		:= FALSE;
		stMachineCurrentState.ManualMode	:= FALSE;
		strMachine							:= 'Ready';				
		IF bButtonRun THEN
			StateIndex := 60;
		END_IF;
		
	60: //Running State
		stMachineCurrentState.Error 		:= FALSE;
		stMachineCurrentState.CheckSafety	:= FALSE;
		stMachineCurrentState.Aborted		:= FALSE;
		stMachineCurrentState.Initialize	:= FALSE;
		stMachineCurrentState.CheckToRun	:= FALSE;
		stMachineCurrentState.Ready			:= FALSE;
		stMachineCurrentState.Running		:= TRUE;
		stMachineCurrentState.Stopped		:= FALSE;
		stMachineCurrentState.ManualMode	:= FALSE;
		strMachine							:= 'Running';		
		IF bButtonStop THEN
			StateIndex := 70;
		END_IF;
		
	70: //Stopped State
		stMachineCurrentState.Error 		:= FALSE;
		stMachineCurrentState.CheckSafety	:= FALSE;
		stMachineCurrentState.Aborted		:= FALSE;
		stMachineCurrentState.Initialize	:= FALSE;
		stMachineCurrentState.CheckToRun	:= FALSE;
		stMachineCurrentState.Ready			:= FALSE;
		stMachineCurrentState.Running		:= FALSE;
		stMachineCurrentState.Stopped		:= TRUE;
		stMachineCurrentState.ManualMode	:= FALSE;
		strMachine							:= 'Stopped';
		IF bButtonRun THEN
			StateIndex := 60;
		END_IF;
		
	1000: //Manual mode operation state
		stMachineCurrentState.Error 		:= FALSE;
		stMachineCurrentState.CheckSafety	:= FALSE;
		stMachineCurrentState.Aborted		:= FALSE;
		stMachineCurrentState.Initialize	:= FALSE;
		stMachineCurrentState.CheckToRun	:= FALSE;
		stMachineCurrentState.Ready			:= FALSE;
		stMachineCurrentState.Running		:= FALSE;
		stMachineCurrentState.Stopped		:= FALSE;
		stMachineCurrentState.ManualMode	:= TRUE;
		strMachine							:= 'Manual';
		IF bFL_AutoModeActive THEN
			StateIndex := 0;
		END_IF
END_CASE;

END_FUNCTION_BLOCK

// ---- POUs/S01_Box/EM01_BoxShorting.TcPOU
PROGRAM EM01_BoxShorting
VAR
//----Motor-----
	//Barecode Reading	
	FB_BarecodeReadingConv				: MotorManagement;
	stBarecodeReadingConv				: stMotor;
	BarecodeReadingConv_ErrorID			: UINT;
	BarecodeReadingConv_Error			: BOOL;
	bFL_BarecodeReadingConv_Forward		: BOOL;
	//Box Infeed Roller Conveyor 1	
	FB_InfeedRollerConv_1				: MotorManagement;
	stInfeedRollerConv_1				: stMotor;
	InfeedRollerConv_1_ErrorID			: UINT;
	InfeedRollerConv_1_Error			: BOOL;
	bFL_InfeedRollerConv_1_Forward		: BOOL;
	//Box Infeed Roller Conveyor 2	
	FB_InfeedRollerConv_2				: MotorManagement;
	stInfeedRollerConv_2				: stMotor;
	InfeedRollerConv_2_ErrorID			: UINT;
	InfeedRollerConv_2_Error			: BOOL;
	bFL_InfeedRollerConv_2_Forward		: BOOL;
	//Box Infeed Roller Conveyor 3	
	FB_InfeedRollerConv_3				: MotorManagement;
	stInfeedRollerConv_3				: stMotor;
	InfeedRollerConv_3_ErrorID			: UINT;
	InfeedRollerConv_3_Error			: BOOL;
	bFL_InfeedRollerConv_3_Forward		: BOOL;
//----Pneumatic-----
	//Box Pusher for Reject Barcode	
	FB_BoxPusherRejectBarcode			: Pneumatic_1Coil_Management;
	stBoxPusherRejectBarcode			: stPneumatic1;
	BoxPusherRejectBarcode_Error		: BOOL;
	BoxPusherRejectBarcode_ErrorID		: INT;
	BoxPusherRejectBarcode_ErrorMsg		: STRING;
	bFL_BoxPusherRejectBarcode_Adv		: BOOL;
	//Box Pusher for Reject Weight	
	FB_BoxPusherRejectWeight			: Pneumatic_1Coil_Management;
	stBoxPusherRejectWeight				: stPneumatic1;
	BoxPusherRejectWeight_Error			: BOOL;
	BoxPusherRejectWeight_ErrorID		: INT;
	BoxPusherRejectWeight_ErrorMsg		: STRING;
	bFL_BoxPusherRejectWeight_Adv		: BOOL;
	//Box Pusher for Robot	
	FB_BoxPusherRobot					: Pneumatic_1Coil_Management;
	stBoxPusherRobot					: stPneumatic1;
	BoxPusherRobot_Error				: BOOL;
	BoxPusherRobot_ErrorID				: INT;
	BoxPusherRobot_ErrorMsg				: STRING;
	bFL_BoxPusherRobot_Adv				: BOOL;
END_VAR

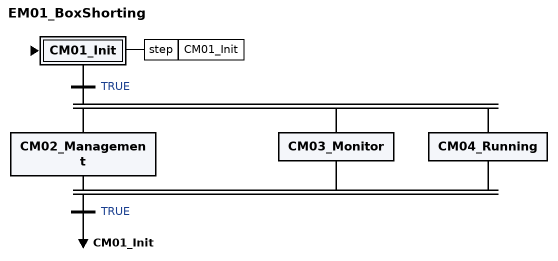
INITIAL_STEP CM01_Init:
    CM01_Init(N);  // step action
END_STEP
TRANSITION FROM CM01_Init TO (CM02_Management, CM03_Monitor, CM04_Running)
    := TRUE;
END_TRANSITION
STEP CM02_Management:
END_STEP
STEP CM03_Monitor:
END_STEP
STEP CM04_Running:
END_STEP
TRANSITION FROM (CM02_Management, CM03_Monitor, CM04_Running) TO CM01_Init
    := TRUE;
END_TRANSITION

ACTION CM01_Init:

END_ACTION

ACTION CM02_Management:
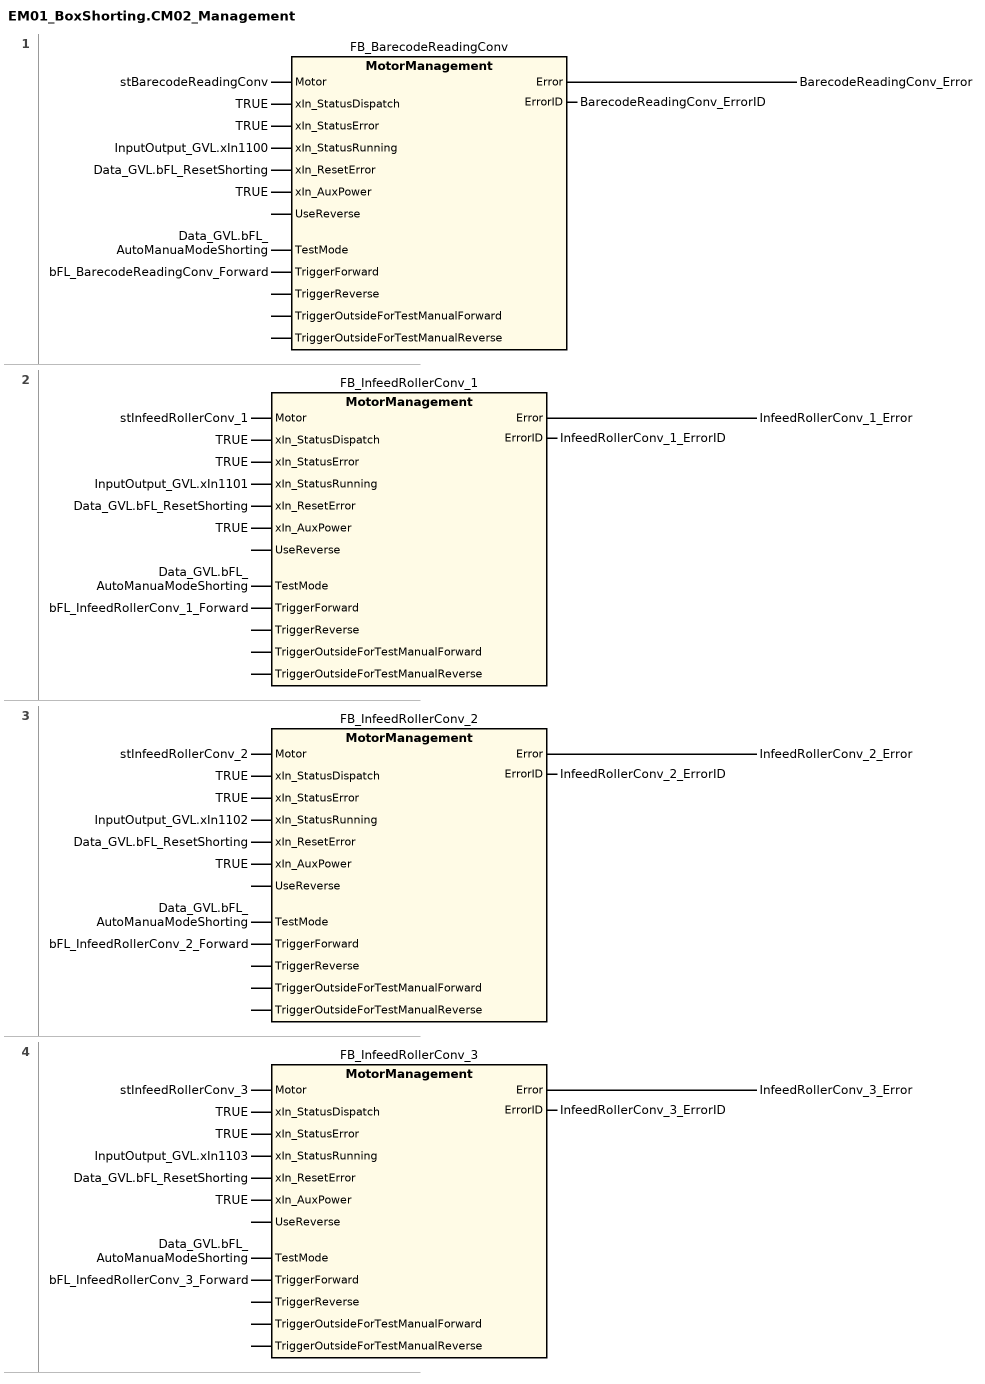
// NETWORK 1
FB_BarecodeReadingConv(
    Motor := stBarecodeReadingConv,
    xIn_StatusDispatch := TRUE,
    xIn_StatusError := TRUE,
    xIn_StatusRunning := InputOutput_GVL.xIn1100,
    xIn_ResetError := Data_GVL.bFL_ResetShorting,
    xIn_AuxPower := TRUE,
    TestMode := Data_GVL.bFL_AutoManuaModeShorting,
    TriggerForward := bFL_BarecodeReadingConv_Forward,
    ErrorID => BarecodeReadingConv_ErrorID); // MotorManagement
BarecodeReadingConv_Error := FB_BarecodeReadingConv.Error;

// NETWORK 2
FB_InfeedRollerConv_1(
    Motor := stInfeedRollerConv_1,
    xIn_StatusDispatch := TRUE,
    xIn_StatusError := TRUE,
    xIn_StatusRunning := InputOutput_GVL.xIn1101,
    xIn_ResetError := Data_GVL.bFL_ResetShorting,
    xIn_AuxPower := TRUE,
    TestMode := Data_GVL.bFL_AutoManuaModeShorting,
    TriggerForward := bFL_InfeedRollerConv_1_Forward,
    ErrorID => InfeedRollerConv_1_ErrorID); // MotorManagement
InfeedRollerConv_1_Error := FB_InfeedRollerConv_1.Error;

// NETWORK 3
FB_InfeedRollerConv_2(
    Motor := stInfeedRollerConv_2,
    xIn_StatusDispatch := TRUE,
    xIn_StatusError := TRUE,
    xIn_StatusRunning := InputOutput_GVL.xIn1102,
    xIn_ResetError := Data_GVL.bFL_ResetShorting,
    xIn_AuxPower := TRUE,
    TestMode := Data_GVL.bFL_AutoManuaModeShorting,
    TriggerForward := bFL_InfeedRollerConv_2_Forward,
    ErrorID => InfeedRollerConv_2_ErrorID); // MotorManagement
InfeedRollerConv_2_Error := FB_InfeedRollerConv_2.Error;

// NETWORK 4
FB_InfeedRollerConv_3(
    Motor := stInfeedRollerConv_3,
    xIn_StatusDispatch := TRUE,
    xIn_StatusError := TRUE,
    xIn_StatusRunning := InputOutput_GVL.xIn1103,
    xIn_ResetError := Data_GVL.bFL_ResetShorting,
    xIn_AuxPower := TRUE,
    TestMode := Data_GVL.bFL_AutoManuaModeShorting,
    TriggerForward := bFL_InfeedRollerConv_3_Forward,
    ErrorID => InfeedRollerConv_3_ErrorID); // MotorManagement
InfeedRollerConv_3_Error := FB_InfeedRollerConv_3.Error;

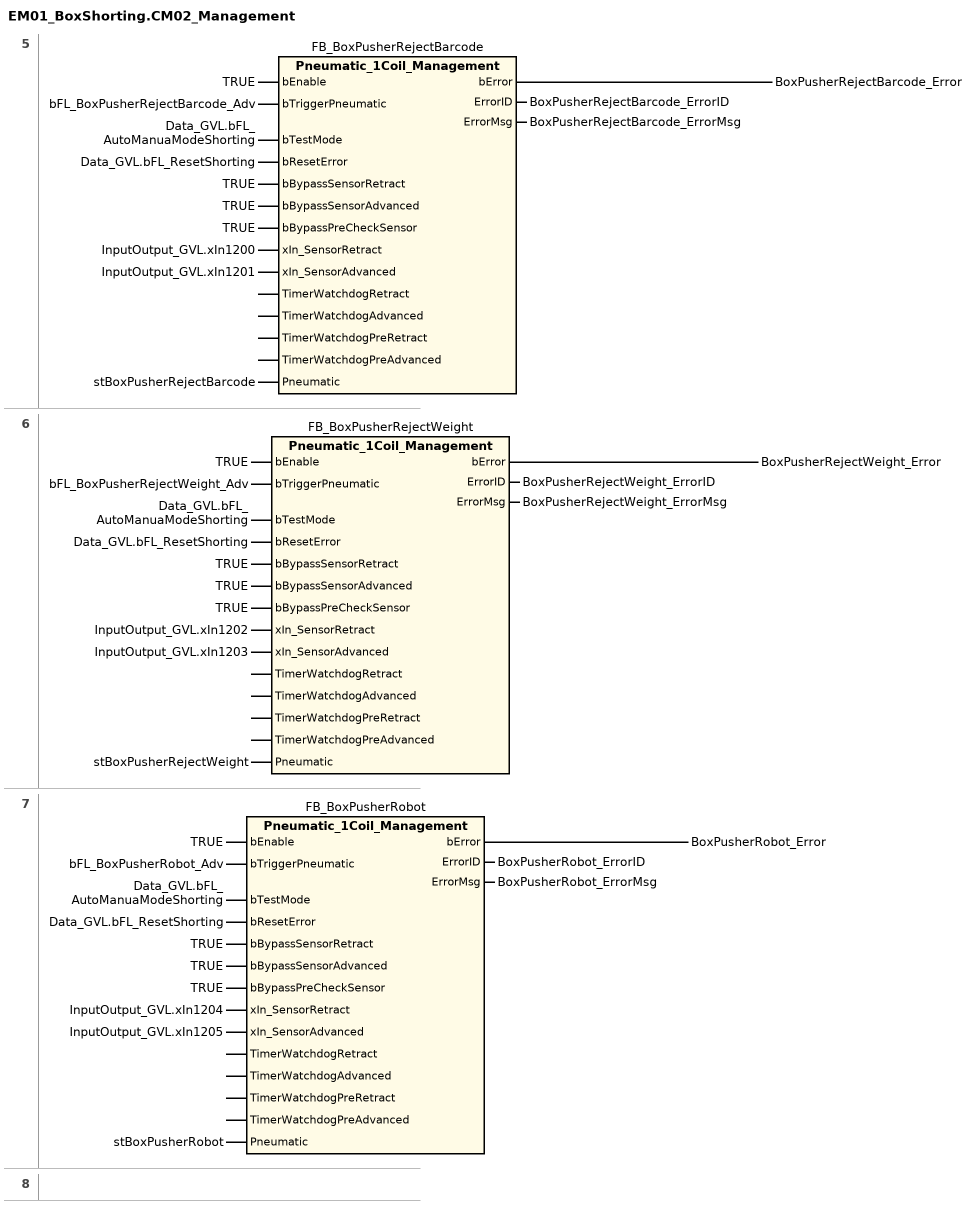
// NETWORK 5
FB_BoxPusherRejectBarcode(
    bEnable := TRUE,
    bTriggerPneumatic := bFL_BoxPusherRejectBarcode_Adv,
    bTestMode := Data_GVL.bFL_AutoManuaModeShorting,
    bResetError := Data_GVL.bFL_ResetShorting,
    bBypassSensorRetract := TRUE,
    bBypassSensorAdvanced := TRUE,
    bBypassPreCheckSensor := TRUE,
    xIn_SensorRetract := InputOutput_GVL.xIn1200,
    xIn_SensorAdvanced := InputOutput_GVL.xIn1201,
    Pneumatic := stBoxPusherRejectBarcode,
    ErrorID => BoxPusherRejectBarcode_ErrorID,
    ErrorMsg => BoxPusherRejectBarcode_ErrorMsg); // Pneumatic_1Coil_Management
BoxPusherRejectBarcode_Error := FB_BoxPusherRejectBarcode.bError;

// NETWORK 6
FB_BoxPusherRejectWeight(
    bEnable := TRUE,
    bTriggerPneumatic := bFL_BoxPusherRejectWeight_Adv,
    bTestMode := Data_GVL.bFL_AutoManuaModeShorting,
    bResetError := Data_GVL.bFL_ResetShorting,
    bBypassSensorRetract := TRUE,
    bBypassSensorAdvanced := TRUE,
    bBypassPreCheckSensor := TRUE,
    xIn_SensorRetract := InputOutput_GVL.xIn1202,
    xIn_SensorAdvanced := InputOutput_GVL.xIn1203,
    Pneumatic := stBoxPusherRejectWeight,
    ErrorID => BoxPusherRejectWeight_ErrorID,
    ErrorMsg => BoxPusherRejectWeight_ErrorMsg); // Pneumatic_1Coil_Management
BoxPusherRejectWeight_Error := FB_BoxPusherRejectWeight.bError;

// NETWORK 7
FB_BoxPusherRobot(
    bEnable := TRUE,
    bTriggerPneumatic := bFL_BoxPusherRobot_Adv,
    bTestMode := Data_GVL.bFL_AutoManuaModeShorting,
    bResetError := Data_GVL.bFL_ResetShorting,
    bBypassSensorRetract := TRUE,
    bBypassSensorAdvanced := TRUE,
    bBypassPreCheckSensor := TRUE,
    xIn_SensorRetract := InputOutput_GVL.xIn1204,
    xIn_SensorAdvanced := InputOutput_GVL.xIn1205,
    Pneumatic := stBoxPusherRobot,
    ErrorID => BoxPusherRobot_ErrorID,
    ErrorMsg => BoxPusherRobot_ErrorMsg); // Pneumatic_1Coil_Management
BoxPusherRobot_Error := FB_BoxPusherRobot.bError;

// NETWORK 8
END_ACTION

ACTION CM03_Monitor:
// NETWORK 1
END_ACTION

ACTION CM04_Running:
// NETWORK 1
END_ACTION

END_PROGRAM

// ---- POUs/Functions Blocks/MotorManagement.TcPOU
FUNCTION_BLOCK MotorManagement
VAR_IN_OUT
	Motor	: stMotor;
END_VAR

VAR_INPUT
	xIn_StatusDispatch: BOOL;
	xIn_StatusError		: BOOL;
	xIn_StatusRunning	: BOOL;
	xIn_ResetError		: BOOL;
	xIn_AuxPower		: BOOL;
	UseReverse			: BOOL;
	TestMode			: BOOL;
	TriggerForward		: BOOL;
	TriggerReverse		: BOOL;
	TriggerOutsideForTestManualForward: BOOL;
	TriggerOutsideForTestManualReverse: BOOL;
END_VAR
VAR_OUTPUT
	Error	: BOOL;
	ErrorID	: UINT;
END_VAR
VAR
	StatusError			: BOOL;
	MotorCannotRunning	: BOOL;
	PowerOff			: BOOL;
	Timer				: TON;
	LocalSwitch_Off		: BOOL;
END_VAR
VAR // added by the converter: edge detectors and wires of the graphical bodies
    _w1 : BOOL;
END_VAR

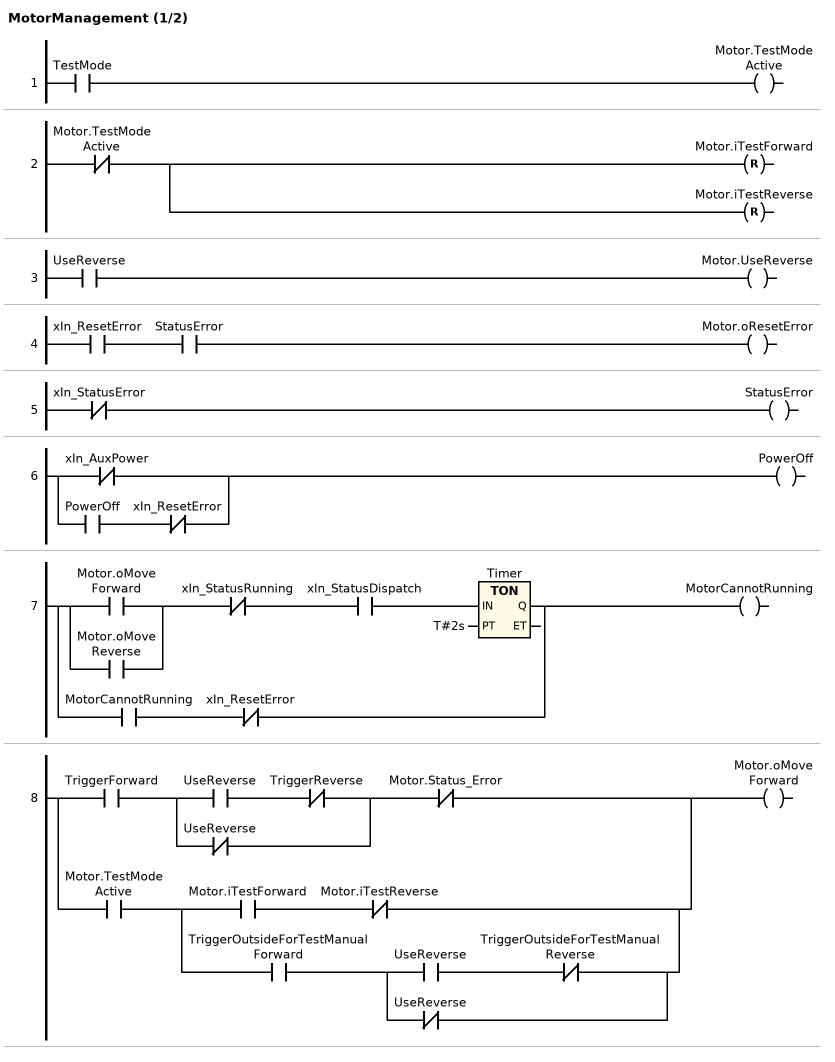
// NETWORK 1
Motor.TestModeActive := TestMode;

// NETWORK 2
_w1 := NOT Motor.TestModeActive;
Motor.iTestForward R= _w1;
Motor.iTestReverse R= _w1;

// NETWORK 3
Motor.UseReverse := UseReverse;

// NETWORK 4
Motor.oResetError := xIn_ResetError AND StatusError;

// NETWORK 5
StatusError := NOT xIn_StatusError;

// NETWORK 6
PowerOff := NOT xIn_AuxPower OR PowerOff AND NOT xIn_ResetError;

// NETWORK 7
Timer(IN := (Motor.oMoveForward OR Motor.oMoveReverse) AND NOT xIn_StatusRunning AND xIn_StatusDispatch, PT := T#2s); // TON
MotorCannotRunning := Timer.Q OR MotorCannotRunning AND NOT xIn_ResetError;

// NETWORK 8
Motor.oMoveForward := TriggerForward AND (UseReverse AND NOT TriggerReverse OR NOT UseReverse) AND NOT Motor.Status_Error OR Motor.TestModeActive AND (Motor.iTestForward AND NOT Motor.iTestReverse OR TriggerOutsideForTestManualForward AND (UseReverse AND NOT TriggerOutsideForTestManualReverse OR NOT UseReverse));

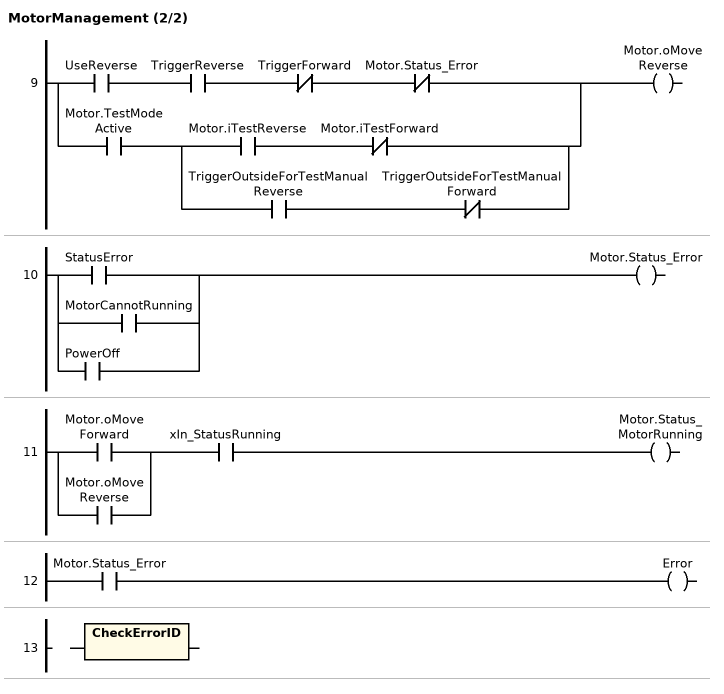
// NETWORK 9
Motor.oMoveReverse := UseReverse AND TriggerReverse AND NOT TriggerForward AND NOT Motor.Status_Error OR Motor.TestModeActive AND (Motor.iTestReverse AND NOT Motor.iTestForward OR TriggerOutsideForTestManualReverse AND NOT TriggerOutsideForTestManualForward);

// NETWORK 10
Motor.Status_Error := StatusError OR MotorCannotRunning OR PowerOff;

// NETWORK 11
Motor.Status_MotorRunning := (Motor.oMoveForward OR Motor.oMoveReverse) AND xIn_StatusRunning;

// NETWORK 12
Error := Motor.Status_Error;

// NETWORK 13
CheckErrorID();

ACTION CheckErrorID:
IF Error THEN
	IF StatusError THEN
		ErrorID:=1;
	ELSIF PowerOff THEN
			ErrorID:=2;
		ELSIF LocalSwitch_Off THEN
				ErrorID:=3;
			ELSIF MotorCannotRunning THEN
					ErrorID:=10;
				ELSE
					ErrorID:=90;
			END_IF
ELSE
	ErrorID:=0;
END_IF

Motor.ErrorID:=ErrorID;
END_ACTION

END_FUNCTION_BLOCK

// ---- POUs/Functions Blocks/Pneumatic_1Coil_Management.TcPOU
FUNCTION_BLOCK Pneumatic_1Coil_Management
// Function block untuk mengolah faceplate dan watchdog pneumatic valve 1 coil
//	UDT dependencies:
	(*  
	1. stPneumatic v1.0 	*)

//	Changelog:
	(* 
	v1.0 [27.12.2021] Start development function block - Fabrilian Asali	*)	

VAR_INPUT
	bEnable						: BOOL;		
	bTriggerPneumatic			: BOOL;
	bTestMode					: BOOL;
	bResetError					: BOOL;
	bBypassSensorRetract		: BOOL;
	bBypassSensorAdvanced		: BOOL;
	bBypassPreCheckSensor		: BOOL;
	xIn_SensorRetract			: BOOL;
	xIn_SensorAdvanced			: BOOL;
	TimerWatchdogRetract		: TIME := T#5S;
	TimerWatchdogAdvanced		: TIME := T#5S;
	TimerWatchdogPreRetract		: TIME := T#5S;
	TimerWatchdogPreAdvanced	: TIME := T#5S;
END_VAR

VAR_OUTPUT
	bError						: BOOL;
	ErrorID						: INT;
	ErrorMsg					: STRING;
END_VAR

VAR_IN_OUT
	Pneumatic					: stPneumatic1;
END_VAR

VAR
	SeqIndex					: INT;
	WatchdogTimer				: TON;
	bTrig_Output				: BOOL;
END_VAR
VAR // added by the converter: edge detectors and wires of the graphical bodies
    _rt1 : R_TRIG;
    _ft1 : F_TRIG;
END_VAR

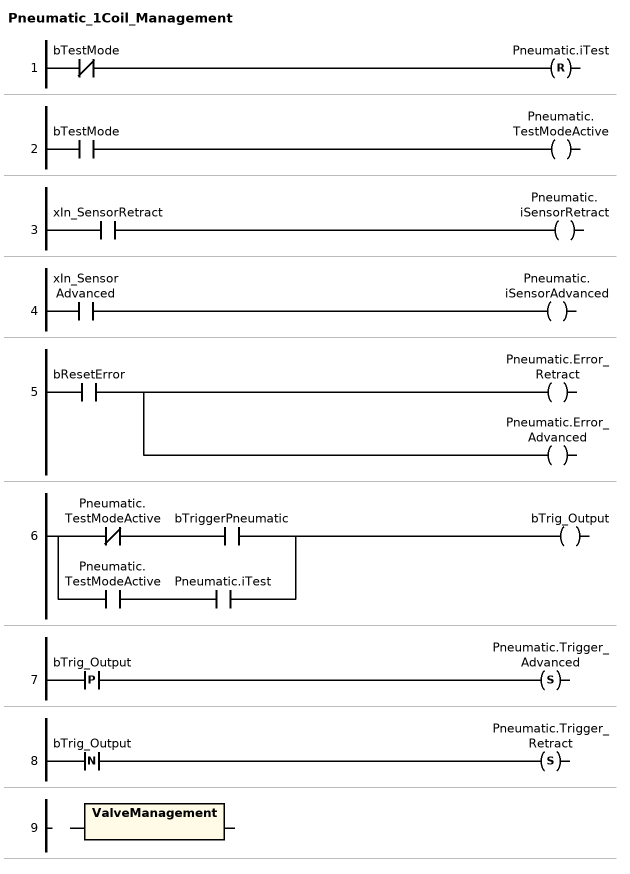
// NETWORK 1
Pneumatic.iTest R= NOT bTestMode;

// NETWORK 2
Pneumatic.TestModeActive := bTestMode;

// NETWORK 3
Pneumatic.iSensorRetract := xIn_SensorRetract;

// NETWORK 4
Pneumatic.iSensorAdvanced := xIn_SensorAdvanced;

// NETWORK 5
Pneumatic.Error_Retract := bResetError;
Pneumatic.Error_Advanced := bResetError;

// NETWORK 6
bTrig_Output := NOT Pneumatic.TestModeActive AND bTriggerPneumatic OR Pneumatic.TestModeActive AND Pneumatic.iTest;

// NETWORK 7
_rt1(CLK := bTrig_Output);
Pneumatic.Trigger_Advanced S= _rt1.Q;

// NETWORK 8
_ft1(CLK := bTrig_Output);
Pneumatic.Trigger_Retract S= _ft1.Q;

// NETWORK 9
ValveManagement();

ACTION ValveManagement:

IF bResetError THEN
	SeqIndex	:= 0;
	ErrorID		:= 0;
	ErrorMsg	:= '';
	bError		:= FALSE;
END_IF

IF bEnable AND NOT bError THEN
	CASE SeqIndex OF
		0:
			IF Pneumatic.Trigger_Retract THEN
				SeqIndex	:= 100;
			ELSIF Pneumatic.Trigger_Advanced THEN
				SeqIndex	:= 200;
			END_IF
		
		100:
			Pneumatic.Trigger_Retract	:= FALSE;
			IF NOT bBypassPreCheckSensor THEN
				WatchdogTimer(In:= TRUE, PT:= TimerWatchdogPreRetract);
				IF Pneumatic.iSensorAdvanced THEN
					WatchdogTimer(In:= FALSE);
					SeqIndex	:= 110;
				ELSIF WatchdogTimer.Q THEN
					WatchdogTimer(In:= FALSE);
					Pneumatic.Error_Retract := TRUE;
					ErrorID					:= 10;
					ErrorMsg				:= 'Error PreCheck Retract';
					SeqIndex	:= 999;
				END_IF
			ELSE
				SeqIndex	:= 110;
			END_IF
	
		110:
			Pneumatic.oPneumatic := FALSE;
			IF NOT bBypassSensorRetract THEN
				WatchdogTimer(In:= TRUE, PT:= TimerWatchdogRetract);
				IF Pneumatic.iSensorRetract THEN
					WatchdogTimer(In:= FALSE);
					SeqIndex	:= 0;
				ELSIF WatchdogTimer.Q THEN
					WatchdogTimer(In:= FALSE);
					Pneumatic.Error_Retract := TRUE;
					ErrorID					:= 11;
					ErrorMsg				:= 'Error Watchdog Retract';
				END_IF
			ELSE
				SeqIndex	:= 0;
			END_IF
			
		200:
			Pneumatic.Trigger_Advanced	:= FALSE;
			IF NOT bBypassPreCheckSensor THEN
				WatchdogTimer(In:= TRUE, PT:= TimerWatchdogPreAdvanced);
				IF Pneumatic.iSensorRetract THEN
					WatchdogTimer(In:= FALSE);
					SeqIndex	:= 210;
				ELSIF WatchdogTimer.Q THEN
					WatchdogTimer(In:= FALSE);
					Pneumatic.Error_Advanced := TRUE;
					ErrorID					:= 20;
					ErrorMsg				:= 'Error PreCheck Advanced';
					SeqIndex	:= 999;
				END_IF
			ELSE
				SeqIndex	:= 210;
			END_IF				
		
		210:
			Pneumatic.oPneumatic := TRUE;
			IF NOT bBypassSensorAdvanced THEN
				WatchdogTimer(In:= TRUE, PT:= TimerWatchdogAdvanced);
				IF Pneumatic.iSensorAdvanced THEN
					WatchdogTimer(In:= FALSE);
					SeqIndex	:= 0;
				ELSIF WatchdogTimer.Q THEN
					WatchdogTimer(In:= FALSE);
					Pneumatic.Error_Advanced := TRUE;
					ErrorID					:= 21;
					ErrorMsg				:= 'Error Watchdog Advanced';
				END_IF
			ELSE
				SeqIndex	:= 0;
			END_IF					
	
		999:
			bError	:= TRUE;	
			
	END_CASE
ELSE
	SeqIndex := 0;
	WatchdogTimer(IN:= FALSE);
	Pneumatic.Trigger_Advanced	:= FALSE;
	Pneumatic.Trigger_Retract	:= FALSE;
END_IF
END_ACTION

END_FUNCTION_BLOCK

// ---- POUs/S02_Pallet/EM01_Dispenser.TcPOU
PROGRAM EM01_Dispenser
VAR
END_VAR

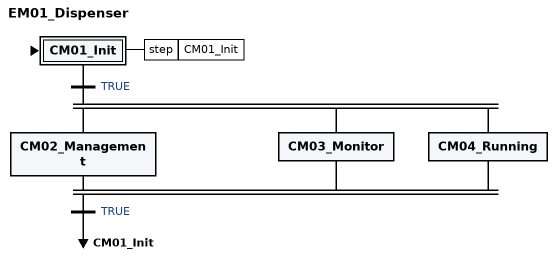
INITIAL_STEP CM01_Init:
    CM01_Init(N);  // step action
END_STEP
TRANSITION FROM CM01_Init TO (CM02_Management, CM03_Monitor, CM04_Running)
    := TRUE;
END_TRANSITION
STEP CM02_Management:
END_STEP
STEP CM03_Monitor:
END_STEP
STEP CM04_Running:
END_STEP
TRANSITION FROM (CM02_Management, CM03_Monitor, CM04_Running) TO CM01_Init
    := TRUE;
END_TRANSITION

ACTION CM01_Init:

END_ACTION

ACTION CM02_Management:
// NETWORK 1
END_ACTION

ACTION CM03_Monitor:
// NETWORK 1
END_ACTION

ACTION CM04_Running:
// NETWORK 1
END_ACTION

END_PROGRAM

// ---- POUs/S02_Pallet/EM02_Shuttle.TcPOU
PROGRAM EM02_Shuttle
VAR
END_VAR

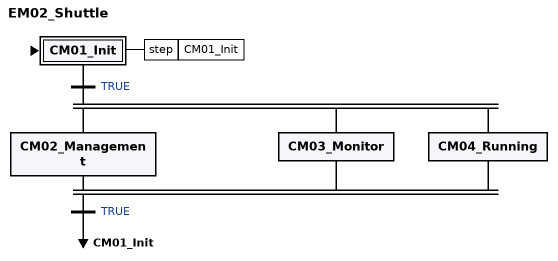
INITIAL_STEP CM01_Init:
    CM01_Init(N);  // step action
END_STEP
TRANSITION FROM CM01_Init TO (CM02_Management, CM03_Monitor, CM04_Running)
    := TRUE;
END_TRANSITION
STEP CM02_Management:
END_STEP
STEP CM03_Monitor:
END_STEP
STEP CM04_Running:
END_STEP
TRANSITION FROM (CM02_Management, CM03_Monitor, CM04_Running) TO CM01_Init
    := TRUE;
END_TRANSITION

ACTION CM01_Init:

END_ACTION

ACTION CM02_Management:
// NETWORK 1
END_ACTION

ACTION CM03_Monitor:
// NETWORK 1
END_ACTION

ACTION CM04_Running:
// NETWORK 1
END_ACTION

END_PROGRAM

// ---- POUs/S02_Pallet/EM03_PalletOutfeed.TcPOU
PROGRAM EM03_PalletOutfeed
VAR
END_VAR

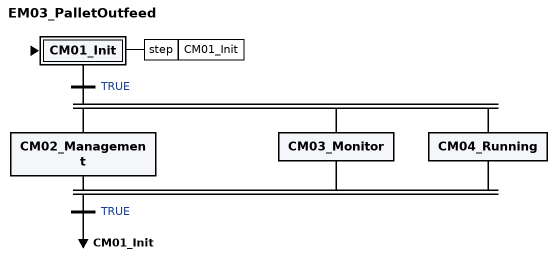
INITIAL_STEP CM01_Init:
    CM01_Init(N);  // step action
END_STEP
TRANSITION FROM CM01_Init TO (CM02_Management, CM03_Monitor, CM04_Running)
    := TRUE;
END_TRANSITION
STEP CM02_Management:
END_STEP
STEP CM03_Monitor:
END_STEP
STEP CM04_Running:
END_STEP
TRANSITION FROM (CM02_Management, CM03_Monitor, CM04_Running) TO CM01_Init
    := TRUE;
END_TRANSITION

ACTION CM01_Init:

END_ACTION

ACTION CM02_Management:
// NETWORK 1
END_ACTION

ACTION CM03_Monitor:
// NETWORK 1
END_ACTION

ACTION CM04_Running:
// NETWORK 1
END_ACTION

END_PROGRAM

// ---- POUs/S02_Pallet/UN01_StateMachinePallet.TcPOU
PROGRAM UN01_StateMachinePallet
VAR
	FB_StateMachineDispenser: FB_StateManager;
	FB_StateMachineShuttle	: FB_StateManager;
	FB_StateMachineOutfeed	: FB_StateManager;
END_VAR

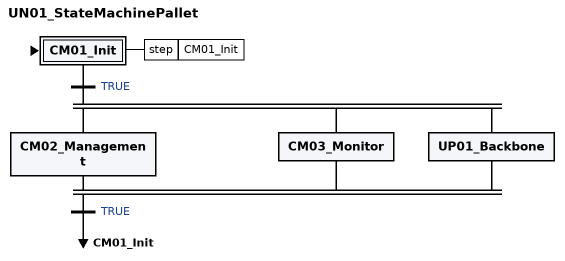
INITIAL_STEP CM01_Init:
    CM01_Init(N);  // step action
END_STEP
TRANSITION FROM CM01_Init TO (CM02_Management, CM03_Monitor, UP01_Backbone)
    := TRUE;
END_TRANSITION
STEP CM02_Management:
END_STEP
STEP CM03_Monitor:
END_STEP
STEP UP01_Backbone:
END_STEP
TRANSITION FROM (CM02_Management, CM03_Monitor, UP01_Backbone) TO CM01_Init
    := TRUE;
END_TRANSITION

ACTION CM01_Init:
//Dispenser
Data_GVL.bFL_StartDispenser 		:= Data_GVL.bStartButton OR HMI_GVL.bStartButtonDispenser;
Data_GVL.bFL_StopDispenser 			:= Data_GVL.bStopButton OR HMI_GVL.bStopButtonDispenser;
Data_GVL.bFL_ResetDispenser 		:= Data_GVL.bResetButton OR HMI_GVL.bResetButtonDispenser;
Data_GVL.bFL_AutoManuaModeDispenser := NOT Data_GVL.StateMachineDispenser.Running AND HMI_GVL.bTestModeEnableDispenser;
//Shuttle
Data_GVL.bFL_StartShuttle 			:= Data_GVL.bStartButton OR HMI_GVL.bStartButtonShuttle;
Data_GVL.bFL_StopShuttle 			:= Data_GVL.bStopButton OR HMI_GVL.bStopButtonShuttle;
Data_GVL.bFL_ResetShuttle 			:= Data_GVL.bResetButton OR HMI_GVL.bResetButtonShuttle;
Data_GVL.bFL_AutoManuaModeShuttle 	:= NOT Data_GVL.StateMachineShuttle.Running AND HMI_GVL.bTestModeEnableShuttle;
//Outfeed
Data_GVL.bFL_StartOutfeed 			:= Data_GVL.bStartButton OR HMI_GVL.bStartButtonOutfeed;
Data_GVL.bFL_StopOutfeed 			:= Data_GVL.bStopButton OR HMI_GVL.bStopButtonOutfeed;
Data_GVL.bFL_ResetOutfeed 			:= Data_GVL.bResetButton OR HMI_GVL.bResetButtonOutfeed;
Data_GVL.bFL_AutoManuaModeOutfeed 	:= NOT Data_GVL.StateMachineOutfeed.Running AND HMI_GVL.bTestModeEnableOutfeed;
END_ACTION

ACTION CM02_Management:
// NETWORK 1
END_ACTION

ACTION CM03_Monitor:
// NETWORK 1
END_ACTION

ACTION UP01_Backbone:
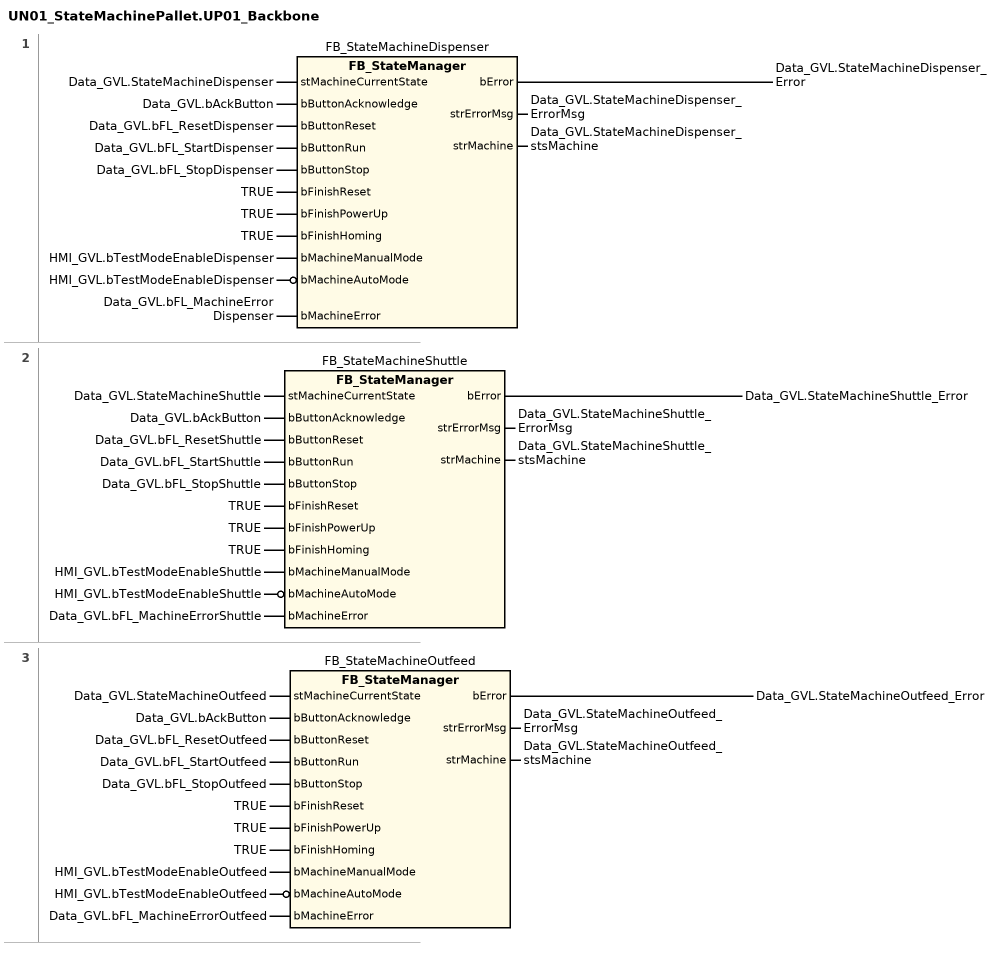
// NETWORK 1
FB_StateMachineDispenser(
    stMachineCurrentState := Data_GVL.StateMachineDispenser,
    bButtonAcknowledge := Data_GVL.bAckButton,
    bButtonReset := Data_GVL.bFL_ResetDispenser,
    bButtonRun := Data_GVL.bFL_StartDispenser,
    bButtonStop := Data_GVL.bFL_StopDispenser,
    bFinishReset := TRUE,
    bFinishPowerUp := TRUE,
    bFinishHoming := TRUE,
    bMachineManualMode := HMI_GVL.bTestModeEnableDispenser,
    bMachineAutoMode := NOT HMI_GVL.bTestModeEnableDispenser,
    bMachineError := Data_GVL.bFL_MachineErrorDispenser,
    strErrorMsg => Data_GVL.StateMachineDispenser_ErrorMsg,
    strMachine => Data_GVL.StateMachineDispenser_stsMachine); // FB_StateManager
Data_GVL.StateMachineDispenser_Error := FB_StateMachineDispenser.bError;

// NETWORK 2
FB_StateMachineShuttle(
    stMachineCurrentState := Data_GVL.StateMachineShuttle,
    bButtonAcknowledge := Data_GVL.bAckButton,
    bButtonReset := Data_GVL.bFL_ResetShuttle,
    bButtonRun := Data_GVL.bFL_StartShuttle,
    bButtonStop := Data_GVL.bFL_StopShuttle,
    bFinishReset := TRUE,
    bFinishPowerUp := TRUE,
    bFinishHoming := TRUE,
    bMachineManualMode := HMI_GVL.bTestModeEnableShuttle,
    bMachineAutoMode := NOT HMI_GVL.bTestModeEnableShuttle,
    bMachineError := Data_GVL.bFL_MachineErrorShuttle,
    strErrorMsg => Data_GVL.StateMachineShuttle_ErrorMsg,
    strMachine => Data_GVL.StateMachineShuttle_stsMachine); // FB_StateManager
Data_GVL.StateMachineShuttle_Error := FB_StateMachineShuttle.bError;

// NETWORK 3
FB_StateMachineOutfeed(
    stMachineCurrentState := Data_GVL.StateMachineOutfeed,
    bButtonAcknowledge := Data_GVL.bAckButton,
    bButtonReset := Data_GVL.bFL_ResetOutfeed,
    bButtonRun := Data_GVL.bFL_StartOutfeed,
    bButtonStop := Data_GVL.bFL_StopOutfeed,
    bFinishReset := TRUE,
    bFinishPowerUp := TRUE,
    bFinishHoming := TRUE,
    bMachineManualMode := HMI_GVL.bTestModeEnableOutfeed,
    bMachineAutoMode := NOT HMI_GVL.bTestModeEnableOutfeed,
    bMachineError := Data_GVL.bFL_MachineErrorOutfeed,
    strErrorMsg => Data_GVL.StateMachineOutfeed_ErrorMsg,
    strMachine => Data_GVL.StateMachineOutfeed_stsMachine); // FB_StateManager
Data_GVL.StateMachineOutfeed_Error := FB_StateMachineOutfeed.bError;
END_ACTION

END_PROGRAM

// ---- POUs/S03_Robot_1/EM03_PlacingArea_2.TcPOU
PROGRAM EM03_PlacingArea_2
VAR
//----Motor-----
	// Box Placing Roller Conveyor 2	
	FB_BoxPlacingRollerConv_2			: MotorManagement;
	stBoxPlacingRollerConv_2			: stMotor;
	BoxPlacingRollerConv_2_ErrorID		: UINT;
	BoxPlacingRollerConv_2_Error		: BOOL;
	bFL_BoxPlacingRollerConv_2_Forward	: BOOL;
	bFL_BoxPlacingRollerConv_2_Reverse	: BOOL;
END_VAR

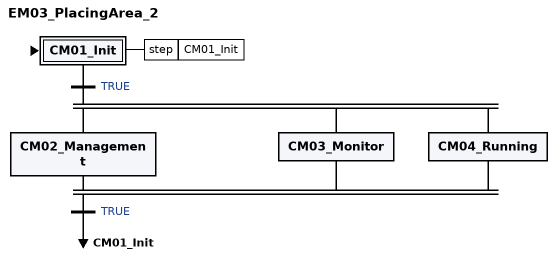
INITIAL_STEP CM01_Init:
    CM01_Init(N);  // step action
END_STEP
TRANSITION FROM CM01_Init TO (CM02_Management, CM03_Monitor, CM04_Running)
    := TRUE;
END_TRANSITION
STEP CM02_Management:
END_STEP
STEP CM03_Monitor:
END_STEP
STEP CM04_Running:
END_STEP
TRANSITION FROM (CM02_Management, CM03_Monitor, CM04_Running) TO CM01_Init
    := TRUE;
END_TRANSITION

ACTION CM01_Init:

END_ACTION

ACTION CM02_Management:
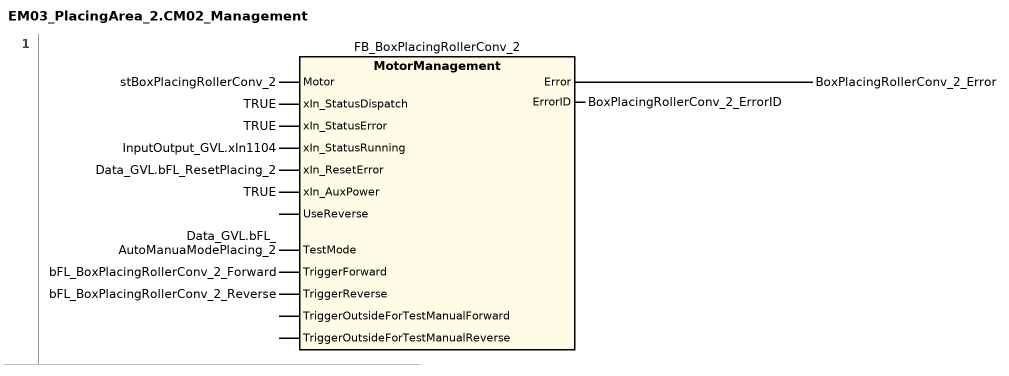
// NETWORK 1
FB_BoxPlacingRollerConv_2(
    Motor := stBoxPlacingRollerConv_2,
    xIn_StatusDispatch := TRUE,
    xIn_StatusError := TRUE,
    xIn_StatusRunning := InputOutput_GVL.xIn1104,
    xIn_ResetError := Data_GVL.bFL_ResetPlacing_2,
    xIn_AuxPower := TRUE,
    TestMode := Data_GVL.bFL_AutoManuaModePlacing_2,
    TriggerForward := bFL_BoxPlacingRollerConv_2_Forward,
    TriggerReverse := bFL_BoxPlacingRollerConv_2_Reverse,
    ErrorID => BoxPlacingRollerConv_2_ErrorID); // MotorManagement
BoxPlacingRollerConv_2_Error := FB_BoxPlacingRollerConv_2.Error;
END_ACTION

ACTION CM03_Monitor:
// NETWORK 1
END_ACTION

ACTION CM04_Running:
// NETWORK 1
END_ACTION

END_PROGRAM

// ---- POUs/S03_Robot_1/EM04_PlacingArea_3.TcPOU
PROGRAM EM04_PlacingArea_3
VAR
//----Motor-----
	// Box Placing Roller Conveyor 3	
	FB_BoxPlacingRollerConv_3			: MotorManagement;
	stBoxPlacingRollerConv_3			: stMotor;
	BoxPlacingRollerConv_3_ErrorID		: UINT;
	BoxPlacingRollerConv_3_Error		: BOOL;
	bFL_BoxPlacingRollerConv_3_Forward	: BOOL;
	bFL_BoxPlacingRollerConv_3_Reverse	: BOOL;
END_VAR

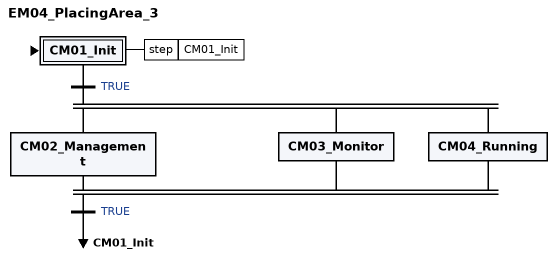
INITIAL_STEP CM01_Init:
    CM01_Init(N);  // step action
END_STEP
TRANSITION FROM CM01_Init TO (CM02_Management, CM03_Monitor, CM04_Running)
    := TRUE;
END_TRANSITION
STEP CM02_Management:
END_STEP
STEP CM03_Monitor:
END_STEP
STEP CM04_Running:
END_STEP
TRANSITION FROM (CM02_Management, CM03_Monitor, CM04_Running) TO CM01_Init
    := TRUE;
END_TRANSITION

ACTION CM01_Init:

END_ACTION

ACTION CM02_Management:
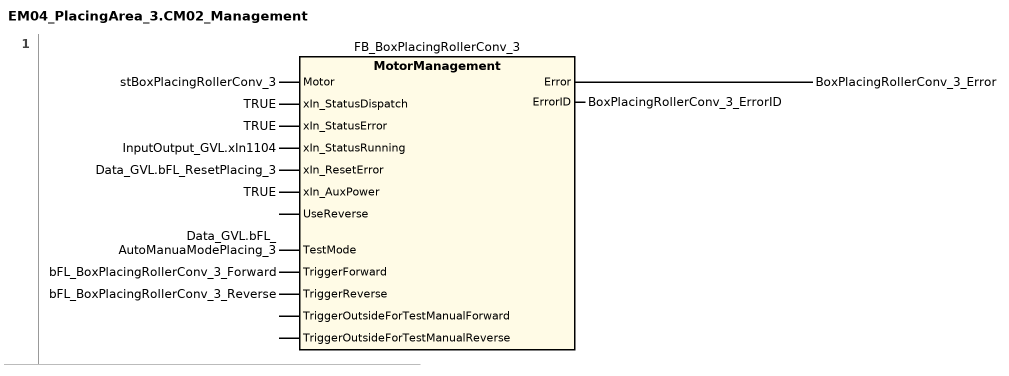
// NETWORK 1
FB_BoxPlacingRollerConv_3(
    Motor := stBoxPlacingRollerConv_3,
    xIn_StatusDispatch := TRUE,
    xIn_StatusError := TRUE,
    xIn_StatusRunning := InputOutput_GVL.xIn1104,
    xIn_ResetError := Data_GVL.bFL_ResetPlacing_3,
    xIn_AuxPower := TRUE,
    TestMode := Data_GVL.bFL_AutoManuaModePlacing_3,
    TriggerForward := bFL_BoxPlacingRollerConv_3_Forward,
    TriggerReverse := bFL_BoxPlacingRollerConv_3_Reverse,
    ErrorID => BoxPlacingRollerConv_3_ErrorID); // MotorManagement
BoxPlacingRollerConv_3_Error := FB_BoxPlacingRollerConv_3.Error;
END_ACTION

ACTION CM03_Monitor:
// NETWORK 1
END_ACTION

ACTION CM04_Running:
// NETWORK 1
END_ACTION

END_PROGRAM

// ---- POUs/S03_Robot_1/EM05_PlacingArea_4.TcPOU
PROGRAM EM05_PlacingArea_4
VAR
//----Motor-----
	// Box Placing Roller Conveyor 4	
	FB_BoxPlacingRollerConv_4					: MotorManagement;
	stBoxPlacingRollerConv_4					: stMotor;
	BoxPlacingRollerConv_4_ErrorID				: UINT;
	BoxPlacingRollerConv_4_Error				: BOOL;
	bFL_BoxPlacingRollerConv_4_Forward			: BOOL;
	bFL_BoxPlacingRollerConv_4_Reverse			: BOOL;
	// Empty And Load Transfer Roller Conveyor 	
	FB_EmptyAndLoadTransferRollerConv			: MotorManagement;
	stEmptyAndLoadTransferRollerConv			: stMotor;
	EmptyAndLoadTransferRollerConv_ErrorID		: UINT;
	EmptyAndLoadTransferRollerConv_Error		: BOOL;
	bFL_EmptyAndLoadTransferRollerConv_Forward	: BOOL;
	bFL_EmptyAndLoadTransferRollerConv_Reverse	: BOOL;
	// Empty And Load Turning Conveyor 1	
	FB_EmptyAndLoadTurningConv_1				: MotorManagement;
	stEmptyAndLoadTurningConv_1					: stMotor;
	EmptyAndLoadTurningConv_1_ErrorID			: UINT;
	EmptyAndLoadTurningConv_1_Error				: BOOL;
	bFL_EmptyAndLoadTurningConv_1_Forward		: BOOL;
	bFL_EmptyAndLoadTurningConv_1_Reverse		: BOOL;
	// Empty And Load Turning Conveyor 2	
	FB_EmptyAndLoadTurningConv_2				: MotorManagement;
	stEmptyAndLoadTurningConv_2					: stMotor;
	EmptyAndLoadTurningConv_2_ErrorID			: UINT;
	EmptyAndLoadTurningConv_2_Error				: BOOL;
	bFL_EmptyAndLoadTurningConv_2_Forward		: BOOL;
	bFL_EmptyAndLoadTurningConv_2_Reverse		: BOOL;
END_VAR

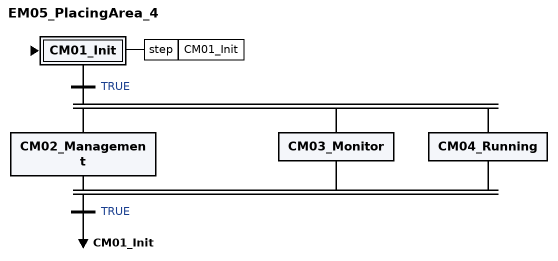
INITIAL_STEP CM01_Init:
    CM01_Init(N);  // step action
END_STEP
TRANSITION FROM CM01_Init TO (CM02_Management, CM03_Monitor, CM04_Running)
    := TRUE;
END_TRANSITION
STEP CM02_Management:
END_STEP
STEP CM03_Monitor:
END_STEP
STEP CM04_Running:
END_STEP
TRANSITION FROM (CM02_Management, CM03_Monitor, CM04_Running) TO CM01_Init
    := TRUE;
END_TRANSITION

ACTION CM01_Init:

END_ACTION

ACTION CM02_Management:
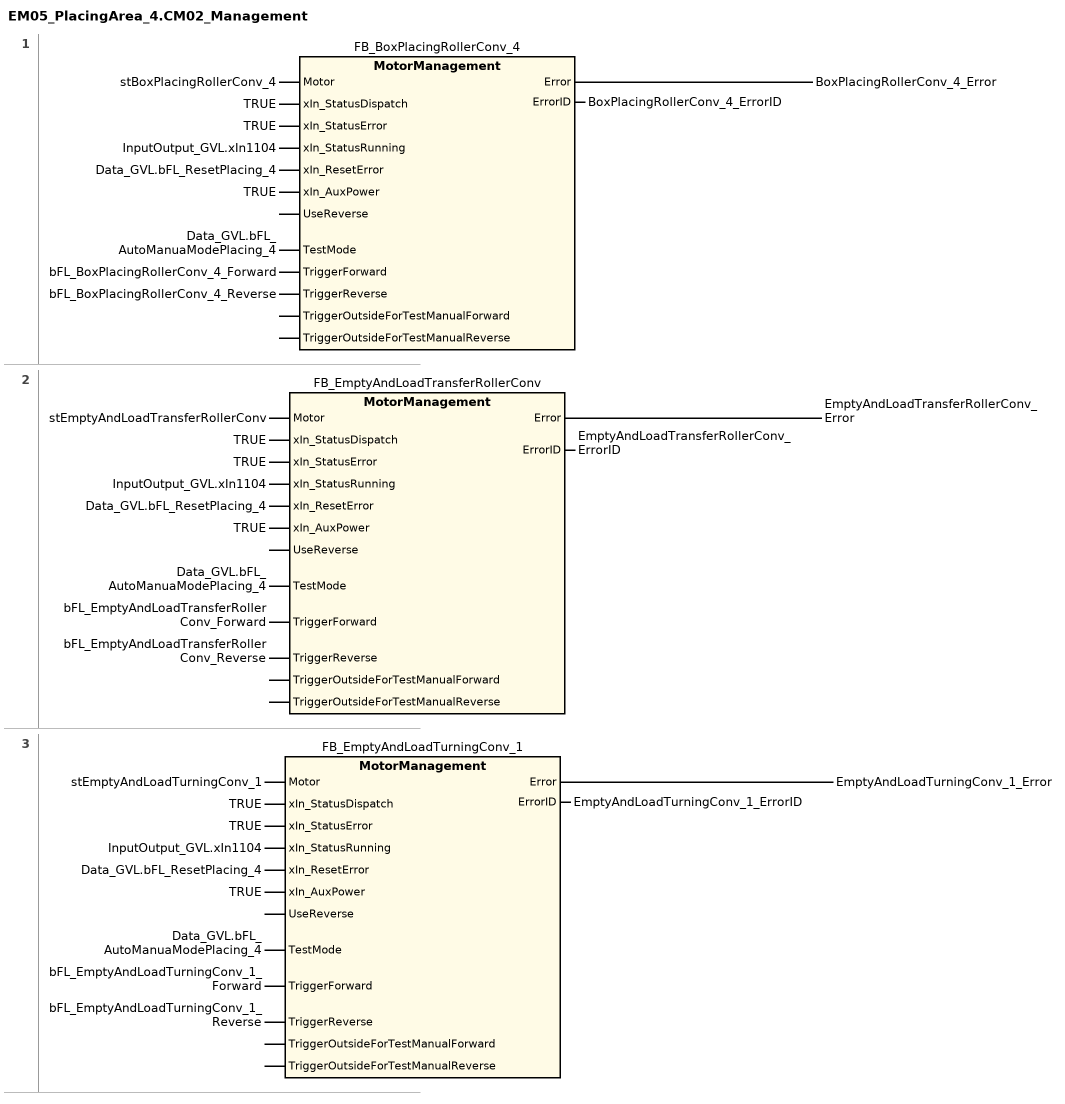
// NETWORK 1
FB_BoxPlacingRollerConv_4(
    Motor := stBoxPlacingRollerConv_4,
    xIn_StatusDispatch := TRUE,
    xIn_StatusError := TRUE,
    xIn_StatusRunning := InputOutput_GVL.xIn1104,
    xIn_ResetError := Data_GVL.bFL_ResetPlacing_4,
    xIn_AuxPower := TRUE,
    TestMode := Data_GVL.bFL_AutoManuaModePlacing_4,
    TriggerForward := bFL_BoxPlacingRollerConv_4_Forward,
    TriggerReverse := bFL_BoxPlacingRollerConv_4_Reverse,
    ErrorID => BoxPlacingRollerConv_4_ErrorID); // MotorManagement
BoxPlacingRollerConv_4_Error := FB_BoxPlacingRollerConv_4.Error;

// NETWORK 2
FB_EmptyAndLoadTransferRollerConv(
    Motor := stEmptyAndLoadTransferRollerConv,
    xIn_StatusDispatch := TRUE,
    xIn_StatusError := TRUE,
    xIn_StatusRunning := InputOutput_GVL.xIn1104,
    xIn_ResetError := Data_GVL.bFL_ResetPlacing_4,
    xIn_AuxPower := TRUE,
    TestMode := Data_GVL.bFL_AutoManuaModePlacing_4,
    TriggerForward := bFL_EmptyAndLoadTransferRollerConv_Forward,
    TriggerReverse := bFL_EmptyAndLoadTransferRollerConv_Reverse,
    ErrorID => EmptyAndLoadTransferRollerConv_ErrorID); // MotorManagement
EmptyAndLoadTransferRollerConv_Error := FB_EmptyAndLoadTransferRollerConv.Error;

// NETWORK 3
FB_EmptyAndLoadTurningConv_1(
    Motor := stEmptyAndLoadTurningConv_1,
    xIn_StatusDispatch := TRUE,
    xIn_StatusError := TRUE,
    xIn_StatusRunning := InputOutput_GVL.xIn1104,
    xIn_ResetError := Data_GVL.bFL_ResetPlacing_4,
    xIn_AuxPower := TRUE,
    TestMode := Data_GVL.bFL_AutoManuaModePlacing_4,
    TriggerForward := bFL_EmptyAndLoadTurningConv_1_Forward,
    TriggerReverse := bFL_EmptyAndLoadTurningConv_1_Reverse,
    ErrorID => EmptyAndLoadTurningConv_1_ErrorID); // MotorManagement
EmptyAndLoadTurningConv_1_Error := FB_EmptyAndLoadTurningConv_1.Error;

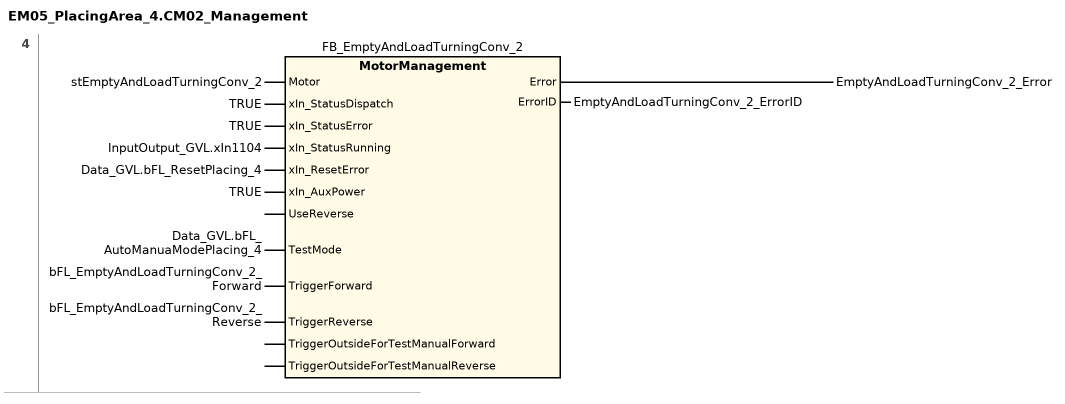
// NETWORK 4
FB_EmptyAndLoadTurningConv_2(
    Motor := stEmptyAndLoadTurningConv_2,
    xIn_StatusDispatch := TRUE,
    xIn_StatusError := TRUE,
    xIn_StatusRunning := InputOutput_GVL.xIn1104,
    xIn_ResetError := Data_GVL.bFL_ResetPlacing_4,
    xIn_AuxPower := TRUE,
    TestMode := Data_GVL.bFL_AutoManuaModePlacing_4,
    TriggerForward := bFL_EmptyAndLoadTurningConv_2_Forward,
    TriggerReverse := bFL_EmptyAndLoadTurningConv_2_Reverse,
    ErrorID => EmptyAndLoadTurningConv_2_ErrorID); // MotorManagement
EmptyAndLoadTurningConv_2_Error := FB_EmptyAndLoadTurningConv_2.Error;
END_ACTION

ACTION CM03_Monitor:
// NETWORK 1
END_ACTION

ACTION CM04_Running:
// NETWORK 1
END_ACTION

END_PROGRAM

// ---- POUs/S03_Robot_1/EM01_BoxInfeed.TcPOU
PROGRAM EM01_BoxInfeed
VAR
//----Motor-----
	// Box Buffer Roller Conveyor 1	
	FB_BoxBufferRollerConv_1			: MotorManagement;
	stBoxBufferRollerConv_1				: stMotor;
	BoxBufferRollerConv_1_ErrorID		: UINT;
	BoxBufferRollerConv_1_Error			: BOOL;
	bFL_BoxBufferRollerConv_1_Forward	: BOOL;
	// Box Buffer Roller Conveyor 2	
	FB_BoxBufferRollerConv_2			: MotorManagement;
	stBoxBufferRollerConv_2				: stMotor;
	BoxBufferRollerConv_2_ErrorID		: UINT;
	BoxBufferRollerConv_2_Error			: BOOL;
	bFL_BoxBufferRollerConv_2_Forward	: BOOL;
	// Box Stop & Go Belt Conveyor
	FB_BoxStopEndGoBeltConv				: MotorManagement;
	stBoxStopEndGoBeltConv				: stMotor;
	BoxStopEndGoBeltConv_ErrorID		: UINT;
	BoxStopEndGoBeltConv_Error			: BOOL;
	bFL_BoxStopEndGoBeltConv_Forward	: BOOL;
	// Box Picking Roller Conveyor
	FB_BoxPickingRollerConv				: MotorManagement;
	stBoxPickingRollerConv				: stMotor;
	BoxPickingRollerConv_ErrorID		: UINT;
	BoxPickingRollerConv_Error			: BOOL;
	bFL_BoxPickingRollerConv_Forward	: BOOL;
END_VAR

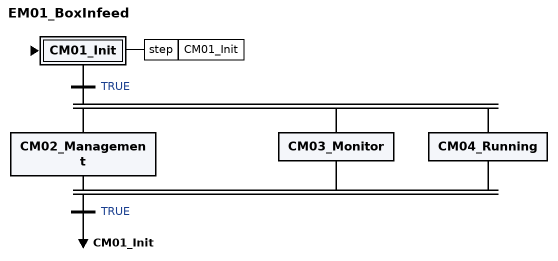
INITIAL_STEP CM01_Init:
    CM01_Init(N);  // step action
END_STEP
TRANSITION FROM CM01_Init TO (CM02_Management, CM03_Monitor, CM04_Running)
    := TRUE;
END_TRANSITION
STEP CM02_Management:
END_STEP
STEP CM03_Monitor:
END_STEP
STEP CM04_Running:
END_STEP
TRANSITION FROM (CM02_Management, CM03_Monitor, CM04_Running) TO CM01_Init
    := TRUE;
END_TRANSITION

ACTION CM01_Init:

END_ACTION

ACTION CM02_Management:
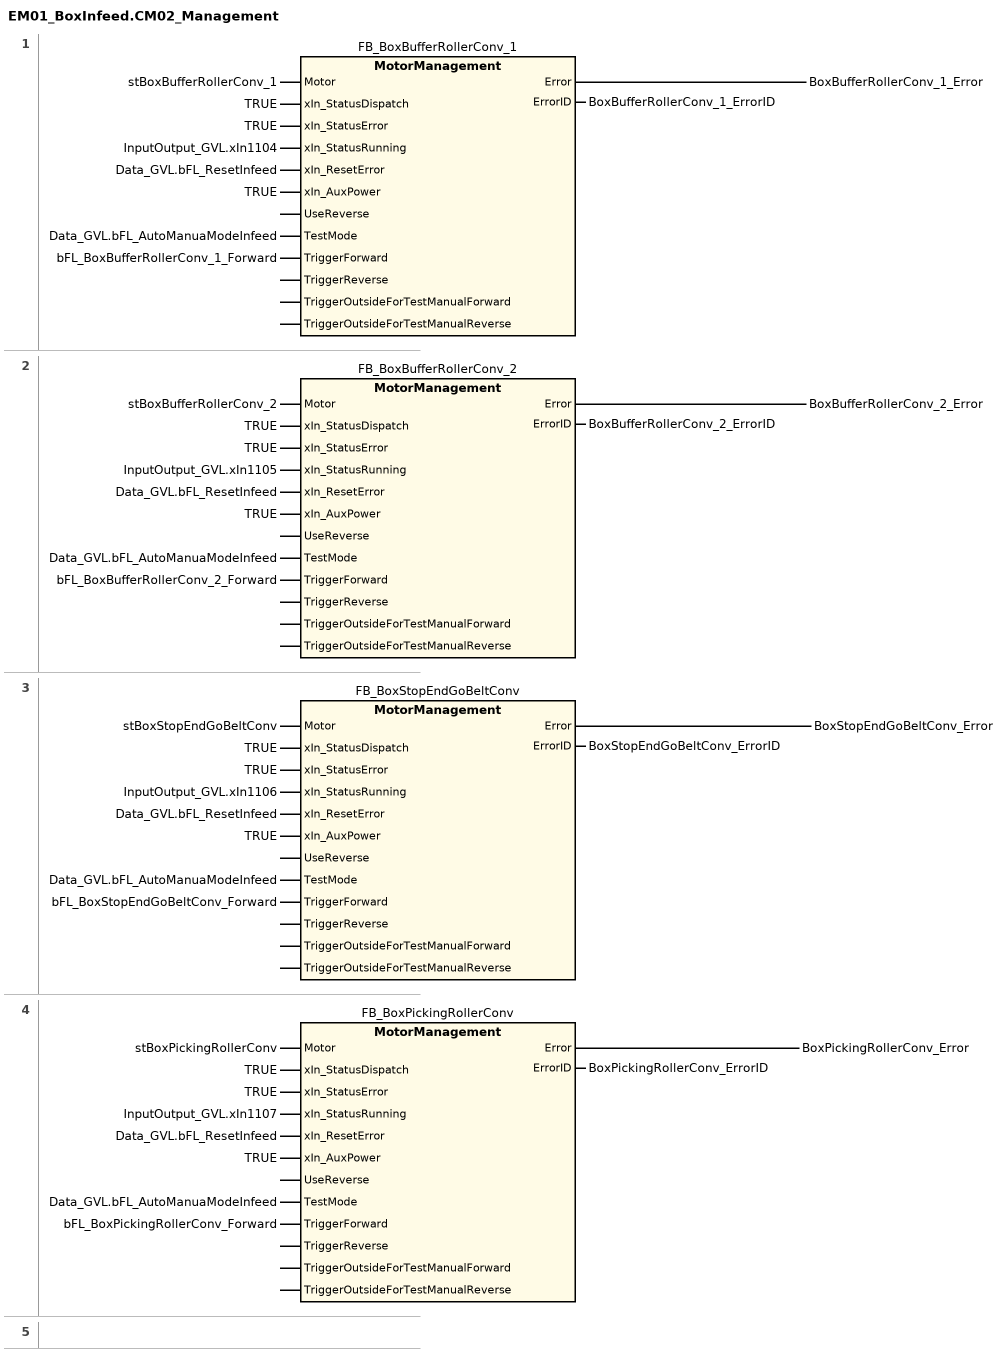
// NETWORK 1
FB_BoxBufferRollerConv_1(
    Motor := stBoxBufferRollerConv_1,
    xIn_StatusDispatch := TRUE,
    xIn_StatusError := TRUE,
    xIn_StatusRunning := InputOutput_GVL.xIn1104,
    xIn_ResetError := Data_GVL.bFL_ResetInfeed,
    xIn_AuxPower := TRUE,
    TestMode := Data_GVL.bFL_AutoManuaModeInfeed,
    TriggerForward := bFL_BoxBufferRollerConv_1_Forward,
    ErrorID => BoxBufferRollerConv_1_ErrorID); // MotorManagement
BoxBufferRollerConv_1_Error := FB_BoxBufferRollerConv_1.Error;

// NETWORK 2
FB_BoxBufferRollerConv_2(
    Motor := stBoxBufferRollerConv_2,
    xIn_StatusDispatch := TRUE,
    xIn_StatusError := TRUE,
    xIn_StatusRunning := InputOutput_GVL.xIn1105,
    xIn_ResetError := Data_GVL.bFL_ResetInfeed,
    xIn_AuxPower := TRUE,
    TestMode := Data_GVL.bFL_AutoManuaModeInfeed,
    TriggerForward := bFL_BoxBufferRollerConv_2_Forward,
    ErrorID => BoxBufferRollerConv_2_ErrorID); // MotorManagement
BoxBufferRollerConv_2_Error := FB_BoxBufferRollerConv_2.Error;

// NETWORK 3
FB_BoxStopEndGoBeltConv(
    Motor := stBoxStopEndGoBeltConv,
    xIn_StatusDispatch := TRUE,
    xIn_StatusError := TRUE,
    xIn_StatusRunning := InputOutput_GVL.xIn1106,
    xIn_ResetError := Data_GVL.bFL_ResetInfeed,
    xIn_AuxPower := TRUE,
    TestMode := Data_GVL.bFL_AutoManuaModeInfeed,
    TriggerForward := bFL_BoxStopEndGoBeltConv_Forward,
    ErrorID => BoxStopEndGoBeltConv_ErrorID); // MotorManagement
BoxStopEndGoBeltConv_Error := FB_BoxStopEndGoBeltConv.Error;

// NETWORK 4
FB_BoxPickingRollerConv(
    Motor := stBoxPickingRollerConv,
    xIn_StatusDispatch := TRUE,
    xIn_StatusError := TRUE,
    xIn_StatusRunning := InputOutput_GVL.xIn1107,
    xIn_ResetError := Data_GVL.bFL_ResetInfeed,
    xIn_AuxPower := TRUE,
    TestMode := Data_GVL.bFL_AutoManuaModeInfeed,
    TriggerForward := bFL_BoxPickingRollerConv_Forward,
    ErrorID => BoxPickingRollerConv_ErrorID); // MotorManagement
BoxPickingRollerConv_Error := FB_BoxPickingRollerConv.Error;

// NETWORK 5
END_ACTION

ACTION CM03_Monitor:
// NETWORK 1
END_ACTION

ACTION CM04_Running:
// NETWORK 1
END_ACTION

END_PROGRAM

// ---- POUs/S03_Robot_1/EM02_PlacingArea_1.TcPOU
PROGRAM EM02_PlacingArea_1
VAR
//----Motor-----
	// Box Placing Roller Conveyor 1	
	FB_BoxPlacingRollerConv_1			: MotorManagement;
	stBoxPlacingRollerConv_1			: stMotor;
	BoxPlacingRollerConv_1_ErrorID		: UINT;
	BoxPlacingRollerConv_1_Error		: BOOL;
	bFL_BoxPlacingRollerConv_1_Forward	: BOOL;
	bFL_BoxPlacingRollerConv_1_Reverse	: BOOL;
END_VAR

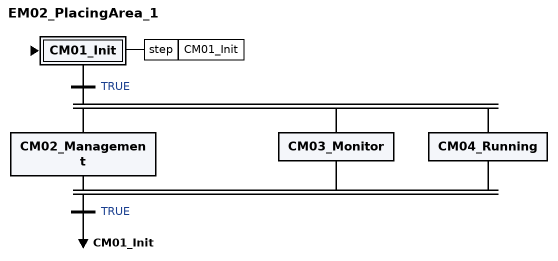
INITIAL_STEP CM01_Init:
    CM01_Init(N);  // step action
END_STEP
TRANSITION FROM CM01_Init TO (CM02_Management, CM03_Monitor, CM04_Running)
    := TRUE;
END_TRANSITION
STEP CM02_Management:
END_STEP
STEP CM03_Monitor:
END_STEP
STEP CM04_Running:
END_STEP
TRANSITION FROM (CM02_Management, CM03_Monitor, CM04_Running) TO CM01_Init
    := TRUE;
END_TRANSITION

ACTION CM01_Init:

END_ACTION

ACTION CM02_Management:
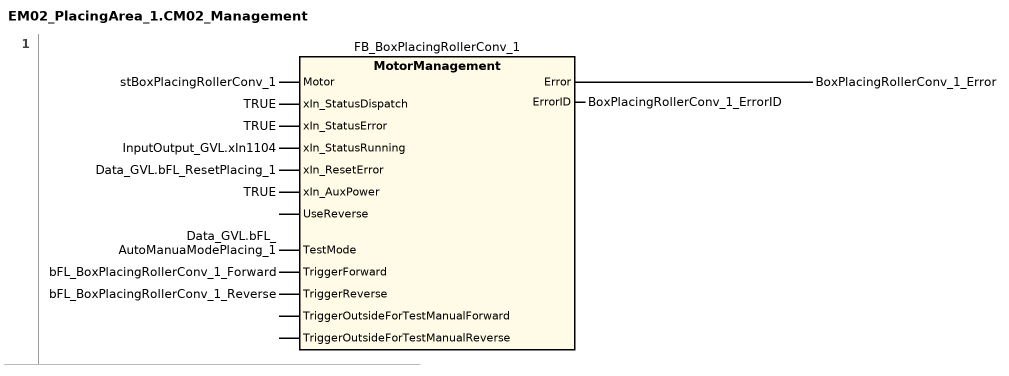
// NETWORK 1
FB_BoxPlacingRollerConv_1(
    Motor := stBoxPlacingRollerConv_1,
    xIn_StatusDispatch := TRUE,
    xIn_StatusError := TRUE,
    xIn_StatusRunning := InputOutput_GVL.xIn1104,
    xIn_ResetError := Data_GVL.bFL_ResetPlacing_1,
    xIn_AuxPower := TRUE,
    TestMode := Data_GVL.bFL_AutoManuaModePlacing_1,
    TriggerForward := bFL_BoxPlacingRollerConv_1_Forward,
    TriggerReverse := bFL_BoxPlacingRollerConv_1_Reverse,
    ErrorID => BoxPlacingRollerConv_1_ErrorID); // MotorManagement
BoxPlacingRollerConv_1_Error := FB_BoxPlacingRollerConv_1.Error;
END_ACTION

ACTION CM03_Monitor:
// NETWORK 1
END_ACTION

ACTION CM04_Running:
// NETWORK 1
END_ACTION

END_PROGRAM

// ---- POUs/S03_Robot_1/EM06_Robot.TcPOU
PROGRAM EM06_Robot
VAR
END_VAR

